gfCNCPoint3[24009] = {X 169.4126, Y 35.0505, Z -4.6667, A 0.000, B 0.000, C 0.000 }
gfCNCPoint3[24010] = {X 169.5555, Y 33.2588, Z -4.6667, A 0.000, B 0.000, C 0.000 }
gfCNCPoint3[24011] = {X 169.9217, Y 31.4991, Z -4.6667, A 0.000, B 0.000, C 0.000 }
gfCNCPoint3[24012] = {X 170.5055, Y 29.7991, Z -4.6667, A 0.000, B 0.000, C 0.000 }
gfCNCPoint3[24013] = {X 171.2083, Y 28.3890, Z -4.6667, A 0.000, B 0.000, C 0.000 }
gfCNCPoint3[24014] = {X 172.1134, Y 27.0994, Z -4.6667, A 0.000, B 0.000, C 0.000 }
gfCNCPoint3[24015] = {X 173.2007, Y 25.9592, Z -4.6667, A 0.000, B 0.000, C 0.000 }
gfCNCPoint3[24016] = {X 174.4459, Y 24.9938, Z -4.6667, A 0.000, B 0.000, C 0.000 }
gfCNCPoint3[24017] = {X 175.8210, Y 24.2248, Z -4.6667, A 0.000, B 0.000, C 0.000 }
gfCNCPoint3[24018] = {X 175.0301, Y 24.0138, Z -4.6667, A 0.000, B 0.000, C 0.000 }
gfCNCPoint3[24019] = {X 174.2987, Y 23.6462, Z -4.6667, A 0.000, B 0.000, C 0.000 }
gfCNCPoint3[24020] = {X 173.6575, Y 23.1374, Z -4.6667, A 0.000, B 0.000, C 0.000 }
gfCNCPoint3[24021] = {X 173.1332, Y 22.5088, Z -4.6667, A 0.000, B 0.000, C 0.000 }
gfCNCPoint3[24022] = {X 172.7479, Y 21.7866, Z -4.6667, A 0.000, B 0.000, C 0.000 }
gfCNCPoint3[24023] = {X 171.4542, Y 18.6179, Z -4.6667, A 0.000, B 0.000, C 0.000 }
gfCNCPoint3[24024] = {X 167.6769, Y 20.1601, Z -4.6667, A 0.000, B 0.000, C 0.000 }
gfCNCPoint3[24025] = {X 167.6769, Y 20.1601, Z -1.6667, A 0.000, B 0.000, C 0.000 }
gfCNCPoint3[24026] = {X 167.6769, Y 20.1601, Z 11.0000, A 0.000, B 0.000, C 0.000 }
gfCNCPoint3[24027] = {X 210.1649, Y 28.5740, Z 11.0000, A 0.000, B 0.000, C 0.000 }
gfCNCPoint3[24028] = {X 210.1649, Y 28.5740, Z -1.6667, A 0.000, B 0.000, C 0.000 }
gfCNCPoint3[24029] = {X 210.1649, Y 28.5740, Z -4.6667, A 0.000, B 0.000, C 0.000 }
gfCNCPoint3[24030] = {X 214.2449, Y 28.5740, Z -4.6667, A 0.000, B 0.000, C 0.000 }
gfCNCPoint3[24031] = {X 214.2449, Y 17.4625, Z -4.6667, A 0.000, B 0.000, C 0.000 }
gfCNCPoint3[24032] = {X 214.2395, Y 16.7693, Z -4.6667, A 0.000, B 0.000, C 0.000 }
gfCNCPoint3[24033] = {X 214.2427, Y 16.2726, Z -4.6667, A 0.000, B 0.000, C 0.000 }
gfCNCPoint3[24034] = {X 213.6048, Y 15.6014, Z -4.6667, A 0.000, B 0.000, C 0.000 }
gfCNCPoint3[24035] = {X 213.1246, Y 14.8098, Z -4.6667, A 0.000, B 0.000, C 0.000 }
gfCNCPoint3[24036] = {X 212.8241, Y 13.9340, Z -4.6667, A 0.000, B 0.000, C 0.000 }
gfCNCPoint3[24037] = {X 212.7172, Y 13.0143, Z -4.6667, A 0.000, B 0.000, C 0.000 }
gfCNCPoint3[24038] = {X 212.7170, Y 12.1868, Z -4.6667, A 0.000, B 0.000, C 0.000 }
gfCNCPoint3[24039] = {X 212.8253, Y 11.2255, Z -4.6667, A 0.000, B 0.000, C 0.000 }
gfCNCPoint3[24040] = {X 213.1448, Y 10.3124, Z -4.6667, A 0.000, B 0.000, C 0.000 }
gfCNCPoint3[24041] = {X 213.6595, Y 9.4933, Z -4.6667, A 0.000, B 0.000, C 0.000 }
gfCNCPoint3[24042] = {X 214.3435, Y 8.8093, Z -4.6667, A 0.000, B 0.000, C 0.000 }
gfCNCPoint3[24043] = {X 215.1626, Y 8.2946, Z -4.6667, A 0.000, B 0.000, C 0.000 }
gfCNCPoint3[24044] = {X 216.0757, Y 7.9751, Z -4.6667, A 0.000, B 0.000, C 0.000 }
gfCNCPoint3[24045] = {X 217.0370, Y 7.8668, Z -4.6667, A 0.000, B 0.000, C 0.000 }
gfCNCPoint3[24046] = {X 223.4805, Y 7.8668, Z -4.6667, A 0.000, B 0.000, C 0.000 }
gfCNCPoint3[24047] = {X 224.4418, Y 7.9751, Z -4.6667, A 0.000, B 0.000, C 0.000 }
gfCNCPoint3[24048] = {X 225.3549, Y 8.2946, Z -4.6667, A 0.000, B 0.000, C 0.000 }
gfCNCPoint3[24049] = {X 226.1740, Y 8.8093, Z -4.6667, A 0.000, B 0.000, C 0.000 }
gfCNCPoint3[24050] = {X 226.8580, Y 9.4933, Z -4.6667, A 0.000, B 0.000, C 0.000 }
gfCNCPoint3[24051] = {X 227.3727, Y 10.3124, Z -4.6667, A 0.000, B 0.000, C 0.000 }
gfCNCPoint3[24052] = {X 227.6922, Y 11.2255, Z -4.6667, A 0.000, B 0.000, C 0.000 }
gfCNCPoint3[24053] = {X 227.8005, Y 12.1868, Z -4.6667, A 0.000, B 0.000, C 0.000 }
gfCNCPoint3[24054] = {X 227.8005, Y 12.9782, Z -4.6667, A 0.000, B 0.000, C 0.000 }
gfCNCPoint3[24055] = {X 227.6992, Y 13.9081, Z -4.6667, A 0.000, B 0.000, C 0.000 }
gfCNCPoint3[24056] = {X 227.4001, Y 14.7944, Z -4.6667, A 0.000, B 0.000, C 0.000 }
gfCNCPoint3[24057] = {X 226.9172, Y 15.5955, Z -4.6667, A 0.000, B 0.000, C 0.000 }
gfCNCPoint3[24058] = {X 226.2732, Y 16.2739, Z -4.6667, A 0.000, B 0.000, C 0.000 }
gfCNCPoint3[24059] = {X 226.2742, Y 40.9155, Z -4.6667, A 0.000, B 0.000, C 0.000 }
gfCNCPoint3[24060] = {X 226.9115, Y 41.5856, Z -4.6667, A 0.000, B 0.000, C 0.000 }
gfCNCPoint3[24061] = {X 227.3916, Y 42.3760, Z -4.6667, A 0.000, B 0.000, C 0.000 }
gfCNCPoint3[24062] = {X 227.6924, Y 43.2504, Z -4.6667, A 0.000, B 0.000, C 0.000 }
gfCNCPoint3[24063] = {X 227.8003, Y 44.1689, Z -4.6667, A 0.000, B 0.000, C 0.000 }
gfCNCPoint3[24064] = {X 227.8005, Y 45.0000, Z -4.6667, A 0.000, B 0.000, C 0.000 }
gfCNCPoint3[24065] = {X 227.6922, Y 45.9613, Z -4.6667, A 0.000, B 0.000, C 0.000 }
gfCNCPoint3[24066] = {X 227.3727, Y 46.8744, Z -4.6667, A 0.000, B 0.000, C 0.000 }
gfCNCPoint3[24067] = {X 226.8580, Y 47.6935, Z -4.6667, A 0.000, B 0.000, C 0.000 }
gfCNCPoint3[24068] = {X 226.1740, Y 48.3775, Z -4.6667, A 0.000, B 0.000, C 0.000 }
gfCNCPoint3[24069] = {X 225.3549, Y 48.8922, Z -4.6667, A 0.000, B 0.000, C 0.000 }
gfCNCPoint3[24070] = {X 224.4418, Y 49.2117, Z -4.6667, A 0.000, B 0.000, C 0.000 }
gfCNCPoint3[24071] = {X 223.4805, Y 49.3200, Z -4.6667, A 0.000, B 0.000, C 0.000 }
gfCNCPoint3[24072] = {X 217.0370, Y 49.3200, Z -4.6667, A 0.000, B 0.000, C 0.000 }
gfCNCPoint3[24073] = {X 216.0805, Y 49.2128, Z -4.6667, A 0.000, B 0.000, C 0.000 }
gfCNCPoint3[24074] = {X 215.1715, Y 48.8964, Z -4.6667, A 0.000, B 0.000, C 0.000 }
gfCNCPoint3[24075] = {X 214.3551, Y 48.3867, Z -4.6667, A 0.000, B 0.000, C 0.000 }
gfCNCPoint3[24076] = {X 213.6718, Y 47.7088, Z -4.6667, A 0.000, B 0.000, C 0.000 }
gfCNCPoint3[24077] = {X 213.1556, Y 46.8965, Z -4.6667, A 0.000, B 0.000, C 0.000 }
gfCNCPoint3[24078] = {X 212.8320, Y 45.9901, Z -4.6667, A 0.000, B 0.000, C 0.000 }
gfCNCPoint3[24079] = {X 212.7172, Y 45.0345, Z -4.6667, A 0.000, B 0.000, C 0.000 }
gfCNCPoint3[24080] = {X 212.7170, Y 44.1958, Z -4.6667, A 0.000, B 0.000, C 0.000 }
gfCNCPoint3[24081] = {X 212.7889, Y 43.4176, Z -4.6667, A 0.000, B 0.000, C 0.000 }
gfCNCPoint3[24082] = {X 213.0019, Y 42.6657, Z -4.6667, A 0.000, B 0.000, C 0.000 }
gfCNCPoint3[24083] = {X 213.3491, Y 41.9656, Z -4.6667, A 0.000, B 0.000, C 0.000 }
gfCNCPoint3[24084] = {X 213.8185, Y 41.3408, Z -4.6667, A 0.000, B 0.000, C 0.000 }
gfCNCPoint3[24085] = {X 214.2405, Y 40.8754, Z -4.6667, A 0.000, B 0.000, C 0.000 }
gfCNCPoint3[24086] = {X 214.2449, Y 40.3061, Z -4.6667, A 0.000, B 0.000, C 0.000 }
gfCNCPoint3[24087] = {X 214.2449, Y 28.5740, Z -4.6667, A 0.000, B 0.000, C 0.000 }
gfCNCPoint3[24088] = {X 210.2449, Y 28.5740, Z -4.6667, A 0.000, B 0.000, C 0.000 }
gfCNCPoint3[24089] = {X 214.3249, Y 28.5740, Z -4.6667, A 0.000, B 0.000, C 0.000 }
gfCNCPoint3[24090] = {X 214.3249, Y 17.4621, Z -4.6667, A 0.000, B 0.000, C 0.000 }
gfCNCPoint3[24091] = {X 214.3195, Y 16.7692, Z -4.6667, A 0.000, B 0.000, C 0.000 }
gfCNCPoint3[24092] = {X 214.3229, Y 16.2355, Z -4.6667, A 0.000, B 0.000, C 0.000 }
gfCNCPoint3[24093] = {X 213.6854, Y 15.5750, Z -4.6667, A 0.000, B 0.000, C 0.000 }
gfCNCPoint3[24094] = {X 213.2050, Y 14.7927, Z -4.6667, A 0.000, B 0.000, C 0.000 }
gfCNCPoint3[24095] = {X 212.9042, Y 13.9254, Z -4.6667, A 0.000, B 0.000, C 0.000 }
gfCNCPoint3[24096] = {X 212.7972, Y 13.0137, Z -4.6667, A 0.000, B 0.000, C 0.000 }
gfCNCPoint3[24097] = {X 212.7970, Y 12.1868, Z -4.6667, A 0.000, B 0.000, C 0.000 }
gfCNCPoint3[24098] = {X 212.9033, Y 11.2433, Z -4.6667, A 0.000, B 0.000, C 0.000 }
gfCNCPoint3[24099] = {X 213.2169, Y 10.3472, Z -4.6667, A 0.000, B 0.000, C 0.000 }
gfCNCPoint3[24100] = {X 213.7220, Y 9.5432, Z -4.6667, A 0.000, B 0.000, C 0.000 }
gfCNCPoint3[24101] = {X 214.3934, Y 8.8719, Z -4.6667, A 0.000, B 0.000, C 0.000 }
gfCNCPoint3[24102] = {X 215.1973, Y 8.3667, Z -4.6667, A 0.000, B 0.000, C 0.000 }
gfCNCPoint3[24103] = {X 216.0935, Y 8.0531, Z -4.6667, A 0.000, B 0.000, C 0.000 }
gfCNCPoint3[24104] = {X 217.0370, Y 7.9468, Z -4.6667, A 0.000, B 0.000, C 0.000 }
gfCNCPoint3[24105] = {X 223.4805, Y 7.9468, Z -4.6667, A 0.000, B 0.000, C 0.000 }
gfCNCPoint3[24106] = {X 224.4240, Y 8.0531, Z -4.6667, A 0.000, B 0.000, C 0.000 }
gfCNCPoint3[24107] = {X 225.3201, Y 8.3667, Z -4.6667, A 0.000, B 0.000, C 0.000 }
gfCNCPoint3[24108] = {X 226.1241, Y 8.8718, Z -4.6667, A 0.000, B 0.000, C 0.000 }
gfCNCPoint3[24109] = {X 226.7954, Y 9.5432, Z -4.6667, A 0.000, B 0.000, C 0.000 }
gfCNCPoint3[24110] = {X 227.3006, Y 10.3471, Z -4.6667, A 0.000, B 0.000, C 0.000 }
gfCNCPoint3[24111] = {X 227.6142, Y 11.2433, Z -4.6667, A 0.000, B 0.000, C 0.000 }
gfCNCPoint3[24112] = {X 227.7205, Y 12.1868, Z -4.6667, A 0.000, B 0.000, C 0.000 }
gfCNCPoint3[24113] = {X 227.7205, Y 12.9781, Z -4.6667, A 0.000, B 0.000, C 0.000 }
gfCNCPoint3[24114] = {X 227.6191, Y 13.8998, Z -4.6667, A 0.000, B 0.000, C 0.000 }
gfCNCPoint3[24115] = {X 227.3197, Y 14.7775, Z -4.6667, A 0.000, B 0.000, C 0.000 }
gfCNCPoint3[24116] = {X 226.8367, Y 15.5690, Z -4.6667, A 0.000, B 0.000, C 0.000 }
gfCNCPoint3[24117] = {X 226.1932, Y 16.2366, Z -4.6667, A 0.000, B 0.000, C 0.000 }
gfCNCPoint3[24118] = {X 226.1942, Y 40.9527, Z -4.6667, A 0.000, B 0.000, C 0.000 }
gfCNCPoint3[24119] = {X 226.8310, Y 41.6122, Z -4.6667, A 0.000, B 0.000, C 0.000 }
gfCNCPoint3[24120] = {X 227.3113, Y 42.3932, Z -4.6667, A 0.000, B 0.000, C 0.000 }
gfCNCPoint3[24121] = {X 227.6124, Y 43.2592, Z -4.6667, A 0.000, B 0.000, C 0.000 }
gfCNCPoint3[24122] = {X 227.7203, Y 44.1697, Z -4.6667, A 0.000, B 0.000, C 0.000 }
gfCNCPoint3[24123] = {X 227.7205, Y 45.0000, Z -4.6667, A 0.000, B 0.000, C 0.000 }
gfCNCPoint3[24124] = {X 227.6142, Y 45.9435, Z -4.6667, A 0.000, B 0.000, C 0.000 }
gfCNCPoint3[24125] = {X 227.3006, Y 46.8397, Z -4.6667, A 0.000, B 0.000, C 0.000 }
gfCNCPoint3[24126] = {X 226.7954, Y 47.6436, Z -4.6667, A 0.000, B 0.000, C 0.000 }
gfCNCPoint3[24127] = {X 226.1241, Y 48.3150, Z -4.6667, A 0.000, B 0.000, C 0.000 }
gfCNCPoint3[24128] = {X 225.3201, Y 48.8201, Z -4.6667, A 0.000, B 0.000, C 0.000 }
gfCNCPoint3[24129] = {X 224.4240, Y 49.1337, Z -4.6667, A 0.000, B 0.000, C 0.000 }
gfCNCPoint3[24130] = {X 223.4805, Y 49.2400, Z -4.6667, A 0.000, B 0.000, C 0.000 }
gfCNCPoint3[24131] = {X 217.0370, Y 49.2400, Z -4.6667, A 0.000, B 0.000, C 0.000 }
gfCNCPoint3[24132] = {X 216.0982, Y 49.1348, Z -4.6667, A 0.000, B 0.000, C 0.000 }
gfCNCPoint3[24133] = {X 215.2061, Y 48.8243, Z -4.6667, A 0.000, B 0.000, C 0.000 }
gfCNCPoint3[24134] = {X 214.4048, Y 48.3240, Z -4.6667, A 0.000, B 0.000, C 0.000 }
gfCNCPoint3[24135] = {X 213.7341, Y 47.6587, Z -4.6667, A 0.000, B 0.000, C 0.000 }
gfCNCPoint3[24136] = {X 213.2275, Y 46.8614, Z -4.6667, A 0.000, B 0.000, C 0.000 }
gfCNCPoint3[24137] = {X 212.9099, Y 45.9717, Z -4.6667, A 0.000, B 0.000, C 0.000 }
gfCNCPoint3[24138] = {X 212.7972, Y 45.0338, Z -4.6667, A 0.000, B 0.000, C 0.000 }
gfCNCPoint3[24139] = {X 212.7970, Y 44.1958, Z -4.6667, A 0.000, B 0.000, C 0.000 }
gfCNCPoint3[24140] = {X 212.8675, Y 43.4322, Z -4.6667, A 0.000, B 0.000, C 0.000 }
gfCNCPoint3[24141] = {X 213.0766, Y 42.6945, Z -4.6667, A 0.000, B 0.000, C 0.000 }
gfCNCPoint3[24142] = {X 213.4172, Y 42.0076, Z -4.6667, A 0.000, B 0.000, C 0.000 }
gfCNCPoint3[24143] = {X 213.8778, Y 41.3946, Z -4.6667, A 0.000, B 0.000, C 0.000 }
gfCNCPoint3[24144] = {X 214.3203, Y 40.9065, Z -4.6667, A 0.000, B 0.000, C 0.000 }
gfCNCPoint3[24145] = {X 214.3249, Y 40.3065, Z -4.6667, A 0.000, B 0.000, C 0.000 }
gfCNCPoint3[24146] = {X 214.3249, Y 28.5740, Z -4.6667, A 0.000, B 0.000, C 0.000 }
gfCNCPoint3[24147] = {X 210.3249, Y 28.5740, Z -4.6667, A 0.000, B 0.000, C 0.000 }
gfCNCPoint3[24148] = {X 214.4049, Y 28.5740, Z -4.6667, A 0.000, B 0.000, C 0.000 }
gfCNCPoint3[24149] = {X 214.4049, Y 17.4618, Z -4.6667, A 0.000, B 0.000, C 0.000 }
gfCNCPoint3[24150] = {X 214.3995, Y 16.7691, Z -4.6667, A 0.000, B 0.000, C 0.000 }
gfCNCPoint3[24151] = {X 214.4031, Y 16.1980, Z -4.6667, A 0.000, B 0.000, C 0.000 }
gfCNCPoint3[24152] = {X 213.7660, Y 15.5482, Z -4.6667, A 0.000, B 0.000, C 0.000 }
gfCNCPoint3[24153] = {X 213.2854, Y 14.7755, Z -4.6667, A 0.000, B 0.000, C 0.000 }
gfCNCPoint3[24154] = {X 212.9843, Y 13.9167, Z -4.6667, A 0.000, B 0.000, C 0.000 }
gfCNCPoint3[24155] = {X 212.8772, Y 13.0130, Z -4.6667, A 0.000, B 0.000, C 0.000 }
gfCNCPoint3[24156] = {X 212.8770, Y 12.1868, Z -4.6667, A 0.000, B 0.000, C 0.000 }
gfCNCPoint3[24157] = {X 212.9813, Y 11.2611, Z -4.6667, A 0.000, B 0.000, C 0.000 }
gfCNCPoint3[24158] = {X 213.2890, Y 10.3819, Z -4.6667, A 0.000, B 0.000, C 0.000 }
gfCNCPoint3[24159] = {X 213.7846, Y 9.5931, Z -4.6667, A 0.000, B 0.000, C 0.000 }
gfCNCPoint3[24160] = {X 214.4433, Y 8.9344, Z -4.6667, A 0.000, B 0.000, C 0.000 }
gfCNCPoint3[24161] = {X 215.2321, Y 8.4388, Z -4.6667, A 0.000, B 0.000, C 0.000 }
gfCNCPoint3[24162] = {X 216.1113, Y 8.1311, Z -4.6667, A 0.000, B 0.000, C 0.000 }
gfCNCPoint3[24163] = {X 217.0370, Y 8.0268, Z -4.6667, A 0.000, B 0.000, C 0.000 }
gfCNCPoint3[24164] = {X 223.4805, Y 8.0268, Z -4.6667, A 0.000, B 0.000, C 0.000 }
gfCNCPoint3[24165] = {X 224.4062, Y 8.1311, Z -4.6667, A 0.000, B 0.000, C 0.000 }
gfCNCPoint3[24166] = {X 225.2854, Y 8.4388, Z -4.6667, A 0.000, B 0.000, C 0.000 }
gfCNCPoint3[24167] = {X 226.0742, Y 8.9344, Z -4.6667, A 0.000, B 0.000, C 0.000 }
gfCNCPoint3[24168] = {X 226.7329, Y 9.5931, Z -4.6667, A 0.000, B 0.000, C 0.000 }
gfCNCPoint3[24169] = {X 227.2285, Y 10.3819, Z -4.6667, A 0.000, B 0.000, C 0.000 }
gfCNCPoint3[24170] = {X 227.5362, Y 11.2611, Z -4.6667, A 0.000, B 0.000, C 0.000 }
gfCNCPoint3[24171] = {X 227.6405, Y 12.1868, Z -4.6667, A 0.000, B 0.000, C 0.000 }
gfCNCPoint3[24172] = {X 227.6405, Y 12.9781, Z -4.6667, A 0.000, B 0.000, C 0.000 }
gfCNCPoint3[24173] = {X 227.5389, Y 13.8916, Z -4.6667, A 0.000, B 0.000, C 0.000 }
gfCNCPoint3[24174] = {X 227.2393, Y 14.7604, Z -4.6667, A 0.000, B 0.000, C 0.000 }
gfCNCPoint3[24175] = {X 226.7562, Y 15.5422, Z -4.6667, A 0.000, B 0.000, C 0.000 }
gfCNCPoint3[24176] = {X 226.1132, Y 16.1989, Z -4.6667, A 0.000, B 0.000, C 0.000 }
gfCNCPoint3[24177] = {X 226.1142, Y 40.9904, Z -4.6667, A 0.000, B 0.000, C 0.000 }
gfCNCPoint3[24178] = {X 226.7506, Y 41.6392, Z -4.6667, A 0.000, B 0.000, C 0.000 }
gfCNCPoint3[24179] = {X 227.2310, Y 42.4107, Z -4.6667, A 0.000, B 0.000, C 0.000 }
gfCNCPoint3[24180] = {X 227.5323, Y 43.2681, Z -4.6667, A 0.000, B 0.000, C 0.000 }
gfCNCPoint3[24181] = {X 227.6403, Y 44.1704, Z -4.6667, A 0.000, B 0.000, C 0.000 }
gfCNCPoint3[24182] = {X 227.6405, Y 45.0000, Z -4.6667, A 0.000, B 0.000, C 0.000 }
gfCNCPoint3[24183] = {X 227.5362, Y 45.9257, Z -4.6667, A 0.000, B 0.000, C 0.000 }
gfCNCPoint3[24184] = {X 227.2285, Y 46.8050, Z -4.6667, A 0.000, B 0.000, C 0.000 }
gfCNCPoint3[24185] = {X 226.7329, Y 47.5937, Z -4.6667, A 0.000, B 0.000, C 0.000 }
gfCNCPoint3[24186] = {X 226.0742, Y 48.2524, Z -4.6667, A 0.000, B 0.000, C 0.000 }
gfCNCPoint3[24187] = {X 225.2854, Y 48.7480, Z -4.6667, A 0.000, B 0.000, C 0.000 }
gfCNCPoint3[24188] = {X 224.4062, Y 49.0557, Z -4.6667, A 0.000, B 0.000, C 0.000 }
gfCNCPoint3[24189] = {X 223.4805, Y 49.1600, Z -4.6667, A 0.000, B 0.000, C 0.000 }
gfCNCPoint3[24190] = {X 217.0370, Y 49.1600, Z -4.6667, A 0.000, B 0.000, C 0.000 }
gfCNCPoint3[24191] = {X 216.1160, Y 49.0568, Z -4.6667, A 0.000, B 0.000, C 0.000 }
gfCNCPoint3[24192] = {X 215.2406, Y 48.7521, Z -4.6667, A 0.000, B 0.000, C 0.000 }
gfCNCPoint3[24193] = {X 214.4544, Y 48.2613, Z -4.6667, A 0.000, B 0.000, C 0.000 }
gfCNCPoint3[24194] = {X 213.7965, Y 47.6085, Z -4.6667, A 0.000, B 0.000, C 0.000 }
gfCNCPoint3[24195] = {X 213.2993, Y 46.8263, Z -4.6667, A 0.000, B 0.000, C 0.000 }
gfCNCPoint3[24196] = {X 212.9877, Y 45.9534, Z -4.6667, A 0.000, B 0.000, C 0.000 }
gfCNCPoint3[24197] = {X 212.8771, Y 45.0332, Z -4.6667, A 0.000, B 0.000, C 0.000 }
gfCNCPoint3[24198] = {X 212.8770, Y 44.1958, Z -4.6667, A 0.000, B 0.000, C 0.000 }
gfCNCPoint3[24199] = {X 212.9461, Y 43.4469, Z -4.6667, A 0.000, B 0.000, C 0.000 }
gfCNCPoint3[24200] = {X 213.1512, Y 42.7233, Z -4.6667, A 0.000, B 0.000, C 0.000 }
gfCNCPoint3[24201] = {X 213.4853, Y 42.0495, Z -4.6667, A 0.000, B 0.000, C 0.000 }
gfCNCPoint3[24202] = {X 213.9370, Y 41.4483, Z -4.6667, A 0.000, B 0.000, C 0.000 }
gfCNCPoint3[24203] = {X 214.4000, Y 40.9376, Z -4.6667, A 0.000, B 0.000, C 0.000 }
gfCNCPoint3[24204] = {X 214.4049, Y 40.3068, Z -4.6667, A 0.000, B 0.000, C 0.000 }
gfCNCPoint3[24205] = {X 214.4049, Y 28.5740, Z -4.6667, A 0.000, B 0.000, C 0.000 }
gfCNCPoint3[24206] = {X 210.4049, Y 28.5740, Z -4.6667, A 0.000, B 0.000, C 0.000 }
gfCNCPoint3[24207] = {X 214.4849, Y 28.5740, Z -4.6667, A 0.000, B 0.000, C 0.000 }
gfCNCPoint3[24208] = {X 214.4849, Y 17.4614, Z -4.6667, A 0.000, B 0.000, C 0.000 }
gfCNCPoint3[24209] = {X 214.4795, Y 16.7691, Z -4.6667, A 0.000, B 0.000, C 0.000 }
gfCNCPoint3[24210] = {X 214.4834, Y 16.1601, Z -4.6667, A 0.000, B 0.000, C 0.000 }
gfCNCPoint3[24211] = {X 214.4254, Y 16.1127, Z -4.6667, A 0.000, B 0.000, C 0.000 }
gfCNCPoint3[24212] = {X 214.3684, Y 16.0642, Z -4.6667, A 0.000, B 0.000, C 0.000 }
gfCNCPoint3[24213] = {X 213.7778, Y 15.4325, Z -4.6667, A 0.000, B 0.000, C 0.000 }
gfCNCPoint3[24214] = {X 213.3338, Y 14.6904, Z -4.6667, A 0.000, B 0.000, C 0.000 }
gfCNCPoint3[24215] = {X 213.0560, Y 13.8714, Z -4.6667, A 0.000, B 0.000, C 0.000 }
gfCNCPoint3[24216] = {X 212.9572, Y 13.0123, Z -4.6667, A 0.000, B 0.000, C 0.000 }
gfCNCPoint3[24217] = {X 212.9570, Y 12.1868, Z -4.6667, A 0.000, B 0.000, C 0.000 }
gfCNCPoint3[24218] = {X 213.0593, Y 11.2789, Z -4.6667, A 0.000, B 0.000, C 0.000 }
gfCNCPoint3[24219] = {X 213.3611, Y 10.4166, Z -4.6667, A 0.000, B 0.000, C 0.000 }
gfCNCPoint3[24220] = {X 213.8471, Y 9.6430, Z -4.6667, A 0.000, B 0.000, C 0.000 }
gfCNCPoint3[24221] = {X 214.4932, Y 8.9969, Z -4.6667, A 0.000, B 0.000, C 0.000 }
gfCNCPoint3[24222] = {X 215.2668, Y 8.5109, Z -4.6667, A 0.000, B 0.000, C 0.000 }
gfCNCPoint3[24223] = {X 216.1291, Y 8.2091, Z -4.6667, A 0.000, B 0.000, C 0.000 }
gfCNCPoint3[24224] = {X 217.0370, Y 8.1068, Z -4.6667, A 0.000, B 0.000, C 0.000 }
gfCNCPoint3[24225] = {X 223.4805, Y 8.1068, Z -4.6667, A 0.000, B 0.000, C 0.000 }
gfCNCPoint3[24226] = {X 224.3884, Y 8.2091, Z -4.6667, A 0.000, B 0.000, C 0.000 }
gfCNCPoint3[24227] = {X 225.2507, Y 8.5109, Z -4.6667, A 0.000, B 0.000, C 0.000 }
gfCNCPoint3[24228] = {X 226.0243, Y 8.9969, Z -4.6667, A 0.000, B 0.000, C 0.000 }
gfCNCPoint3[24229] = {X 226.6704, Y 9.6430, Z -4.6667, A 0.000, B 0.000, C 0.000 }
gfCNCPoint3[24230] = {X 227.1564, Y 10.4166, Z -4.6667, A 0.000, B 0.000, C 0.000 }
gfCNCPoint3[24231] = {X 227.4582, Y 11.2789, Z -4.6667, A 0.000, B 0.000, C 0.000 }
gfCNCPoint3[24232] = {X 227.5605, Y 12.1868, Z -4.6667, A 0.000, B 0.000, C 0.000 }
gfCNCPoint3[24233] = {X 227.5605, Y 12.9781, Z -4.6667, A 0.000, B 0.000, C 0.000 }
gfCNCPoint3[24234] = {X 227.4588, Y 13.8832, Z -4.6667, A 0.000, B 0.000, C 0.000 }
gfCNCPoint3[24235] = {X 227.1589, Y 14.7432, Z -4.6667, A 0.000, B 0.000, C 0.000 }
gfCNCPoint3[24236] = {X 226.6757, Y 15.5152, Z -4.6667, A 0.000, B 0.000, C 0.000 }
gfCNCPoint3[24237] = {X 226.0332, Y 16.1608, Z -4.6667, A 0.000, B 0.000, C 0.000 }
gfCNCPoint3[24238] = {X 226.0342, Y 41.0284, Z -4.6667, A 0.000, B 0.000, C 0.000 }
gfCNCPoint3[24239] = {X 226.1410, Y 41.1156, Z -4.6667, A 0.000, B 0.000, C 0.000 }
gfCNCPoint3[24240] = {X 226.7343, Y 41.7473, Z -4.6667, A 0.000, B 0.000, C 0.000 }
gfCNCPoint3[24241] = {X 227.1808, Y 42.4900, Z -4.6667, A 0.000, B 0.000, C 0.000 }
gfCNCPoint3[24242] = {X 227.4603, Y 43.3103, Z -4.6667, A 0.000, B 0.000, C 0.000 }
gfCNCPoint3[24243] = {X 227.5603, Y 44.1712, Z -4.6667, A 0.000, B 0.000, C 0.000 }
gfCNCPoint3[24244] = {X 227.5605, Y 45.0000, Z -4.6667, A 0.000, B 0.000, C 0.000 }
gfCNCPoint3[24245] = {X 227.4582, Y 45.9079, Z -4.6667, A 0.000, B 0.000, C 0.000 }
gfCNCPoint3[24246] = {X 227.1564, Y 46.7702, Z -4.6667, A 0.000, B 0.000, C 0.000 }
gfCNCPoint3[24247] = {X 226.6704, Y 47.5438, Z -4.6667, A 0.000, B 0.000, C 0.000 }
gfCNCPoint3[24248] = {X 226.0243, Y 48.1899, Z -4.6667, A 0.000, B 0.000, C 0.000 }
gfCNCPoint3[24249] = {X 225.2507, Y 48.6760, Z -4.6667, A 0.000, B 0.000, C 0.000 }
gfCNCPoint3[24250] = {X 224.3884, Y 48.9777, Z -4.6667, A 0.000, B 0.000, C 0.000 }
gfCNCPoint3[24251] = {X 223.4805, Y 49.0800, Z -4.6667, A 0.000, B 0.000, C 0.000 }
gfCNCPoint3[24252] = {X 217.0370, Y 49.0800, Z -4.6667, A 0.000, B 0.000, C 0.000 }
gfCNCPoint3[24253] = {X 216.1337, Y 48.9787, Z -4.6667, A 0.000, B 0.000, C 0.000 }
gfCNCPoint3[24254] = {X 215.2752, Y 48.6800, Z -4.6667, A 0.000, B 0.000, C 0.000 }
gfCNCPoint3[24255] = {X 214.5041, Y 48.1986, Z -4.6667, A 0.000, B 0.000, C 0.000 }
gfCNCPoint3[24256] = {X 213.8588, Y 47.5584, Z -4.6667, A 0.000, B 0.000, C 0.000 }
gfCNCPoint3[24257] = {X 213.3712, Y 46.7912, Z -4.6667, A 0.000, B 0.000, C 0.000 }
gfCNCPoint3[24258] = {X 213.0656, Y 45.9351, Z -4.6667, A 0.000, B 0.000, C 0.000 }
gfCNCPoint3[24259] = {X 212.9571, Y 45.0325, Z -4.6667, A 0.000, B 0.000, C 0.000 }
gfCNCPoint3[24260] = {X 212.9570, Y 44.1958, Z -4.6667, A 0.000, B 0.000, C 0.000 }
gfCNCPoint3[24261] = {X 213.0248, Y 43.4615, Z -4.6667, A 0.000, B 0.000, C 0.000 }
gfCNCPoint3[24262] = {X 213.2259, Y 42.7521, Z -4.6667, A 0.000, B 0.000, C 0.000 }
gfCNCPoint3[24263] = {X 213.5534, Y 42.0915, Z -4.6667, A 0.000, B 0.000, C 0.000 }
gfCNCPoint3[24264] = {X 213.9963, Y 41.5020, Z -4.6667, A 0.000, B 0.000, C 0.000 }
gfCNCPoint3[24265] = {X 214.4798, Y 40.9687, Z -4.6667, A 0.000, B 0.000, C 0.000 }
gfCNCPoint3[24266] = {X 214.4849, Y 40.3072, Z -4.6667, A 0.000, B 0.000, C 0.000 }
gfCNCPoint3[24267] = {X 214.4849, Y 28.5740, Z -4.6667, A 0.000, B 0.000, C 0.000 }
gfCNCPoint3[24268] = {X 210.4849, Y 28.5740, Z -4.6667, A 0.000, B 0.000, C 0.000 }
gfCNCPoint3[24269] = {X 214.5649, Y 28.5740, Z -4.6667, A 0.000, B 0.000, C 0.000 }
gfCNCPoint3[24270] = {X 214.5649, Y 17.4611, Z -4.6667, A 0.000, B 0.000, C 0.000 }
gfCNCPoint3[24271] = {X 214.5595, Y 16.7687, Z -4.6667, A 0.000, B 0.000, C 0.000 }
gfCNCPoint3[24272] = {X 214.5589, Y 16.1867, Z -4.6667, A 0.000, B 0.000, C 0.000 }
gfCNCPoint3[24273] = {X 214.5756, Y 16.1310, Z -4.6667, A 0.000, B 0.000, C 0.000 }
gfCNCPoint3[24274] = {X 214.4973, Y 16.0683, Z -4.6667, A 0.000, B 0.000, C 0.000 }
gfCNCPoint3[24275] = {X 214.4207, Y 16.0037, Z -4.6667, A 0.000, B 0.000, C 0.000 }
gfCNCPoint3[24276] = {X 213.8367, Y 15.3776, Z -4.6667, A 0.000, B 0.000, C 0.000 }
gfCNCPoint3[24277] = {X 213.3993, Y 14.6415, Z -4.6667, A 0.000, B 0.000, C 0.000 }
gfCNCPoint3[24278] = {X 213.1286, Y 13.8292, Z -4.6667, A 0.000, B 0.000, C 0.000 }
gfCNCPoint3[24279] = {X 213.0370, Y 12.9779, Z -4.6667, A 0.000, B 0.000, C 0.000 }
gfCNCPoint3[24280] = {X 213.0370, Y 12.1868, Z -4.6667, A 0.000, B 0.000, C 0.000 }
gfCNCPoint3[24281] = {X 213.1373, Y 11.2967, Z -4.6667, A 0.000, B 0.000, C 0.000 }
gfCNCPoint3[24282] = {X 213.4331, Y 10.4513, Z -4.6667, A 0.000, B 0.000, C 0.000 }
gfCNCPoint3[24283] = {X 213.9097, Y 9.6929, Z -4.6667, A 0.000, B 0.000, C 0.000 }
gfCNCPoint3[24284] = {X 214.5431, Y 9.0595, Z -4.6667, A 0.000, B 0.000, C 0.000 }
gfCNCPoint3[24285] = {X 215.3015, Y 8.5829, Z -4.6667, A 0.000, B 0.000, C 0.000 }
gfCNCPoint3[24286] = {X 216.1469, Y 8.2871, Z -4.6667, A 0.000, B 0.000, C 0.000 }
gfCNCPoint3[24287] = {X 217.0370, Y 8.1868, Z -4.6667, A 0.000, B 0.000, C 0.000 }
gfCNCPoint3[24288] = {X 223.4805, Y 8.1868, Z -4.6667, A 0.000, B 0.000, C 0.000 }
gfCNCPoint3[24289] = {X 224.3706, Y 8.2871, Z -4.6667, A 0.000, B 0.000, C 0.000 }
gfCNCPoint3[24290] = {X 225.2160, Y 8.5829, Z -4.6667, A 0.000, B 0.000, C 0.000 }
gfCNCPoint3[24291] = {X 225.9744, Y 9.0595, Z -4.6667, A 0.000, B 0.000, C 0.000 }
gfCNCPoint3[24292] = {X 226.6078, Y 9.6929, Z -4.6667, A 0.000, B 0.000, C 0.000 }
gfCNCPoint3[24293] = {X 227.0844, Y 10.4513, Z -4.6667, A 0.000, B 0.000, C 0.000 }
gfCNCPoint3[24294] = {X 227.3802, Y 11.2967, Z -4.6667, A 0.000, B 0.000, C 0.000 }
gfCNCPoint3[24295] = {X 227.4805, Y 12.1868, Z -4.6667, A 0.000, B 0.000, C 0.000 }
gfCNCPoint3[24296] = {X 227.4803, Y 13.0192, Z -4.6667, A 0.000, B 0.000, C 0.000 }
gfCNCPoint3[24297] = {X 227.3716, Y 13.9048, Z -4.6667, A 0.000, B 0.000, C 0.000 }
gfCNCPoint3[24298] = {X 227.0694, Y 14.7442, Z -4.6667, A 0.000, B 0.000, C 0.000 }
gfCNCPoint3[24299] = {X 226.5887, Y 15.4958, Z -4.6667, A 0.000, B 0.000, C 0.000 }
gfCNCPoint3[24300] = {X 225.9532, Y 16.1221, Z -4.6667, A 0.000, B 0.000, C 0.000 }
gfCNCPoint3[24301] = {X 225.9542, Y 41.0664, Z -4.6667, A 0.000, B 0.000, C 0.000 }
gfCNCPoint3[24302] = {X 226.0929, Y 41.1797, Z -4.6667, A 0.000, B 0.000, C 0.000 }
gfCNCPoint3[24303] = {X 226.6785, Y 41.8061, Z -4.6667, A 0.000, B 0.000, C 0.000 }
gfCNCPoint3[24304] = {X 227.1171, Y 42.5430, Z -4.6667, A 0.000, B 0.000, C 0.000 }
gfCNCPoint3[24305] = {X 227.3886, Y 43.3563, Z -4.6667, A 0.000, B 0.000, C 0.000 }
gfCNCPoint3[24306] = {X 227.4805, Y 44.2089, Z -4.6667, A 0.000, B 0.000, C 0.000 }
gfCNCPoint3[24307] = {X 227.4805, Y 45.0000, Z -4.6667, A 0.000, B 0.000, C 0.000 }
gfCNCPoint3[24308] = {X 227.3802, Y 45.8901, Z -4.6667, A 0.000, B 0.000, C 0.000 }
gfCNCPoint3[24309] = {X 227.0844, Y 46.7355, Z -4.6667, A 0.000, B 0.000, C 0.000 }
gfCNCPoint3[24310] = {X 226.6078, Y 47.4940, Z -4.6667, A 0.000, B 0.000, C 0.000 }
gfCNCPoint3[24311] = {X 225.9744, Y 48.1273, Z -4.6667, A 0.000, B 0.000, C 0.000 }
gfCNCPoint3[24312] = {X 225.2160, Y 48.6039, Z -4.6667, A 0.000, B 0.000, C 0.000 }
gfCNCPoint3[24313] = {X 224.3706, Y 48.8997, Z -4.6667, A 0.000, B 0.000, C 0.000 }
gfCNCPoint3[24314] = {X 223.4805, Y 49.0000, Z -4.6667, A 0.000, B 0.000, C 0.000 }
gfCNCPoint3[24315] = {X 217.0370, Y 49.0000, Z -4.6667, A 0.000, B 0.000, C 0.000 }
gfCNCPoint3[24316] = {X 216.1469, Y 48.8997, Z -4.6667, A 0.000, B 0.000, C 0.000 }
gfCNCPoint3[24317] = {X 215.3015, Y 48.6039, Z -4.6667, A 0.000, B 0.000, C 0.000 }
gfCNCPoint3[24318] = {X 214.5430, Y 48.1273, Z -4.6667, A 0.000, B 0.000, C 0.000 }
gfCNCPoint3[24319] = {X 213.9097, Y 47.4939, Z -4.6667, A 0.000, B 0.000, C 0.000 }
gfCNCPoint3[24320] = {X 213.4331, Y 46.7355, Z -4.6667, A 0.000, B 0.000, C 0.000 }
gfCNCPoint3[24321] = {X 213.1373, Y 45.8901, Z -4.6667, A 0.000, B 0.000, C 0.000 }
gfCNCPoint3[24322] = {X 213.0370, Y 45.0000, Z -4.6667, A 0.000, B 0.000, C 0.000 }
gfCNCPoint3[24323] = {X 213.0370, Y 44.1958, Z -4.6667, A 0.000, B 0.000, C 0.000 }
gfCNCPoint3[24324] = {X 213.1549, Y 43.2405, Z -4.6667, A 0.000, B 0.000, C 0.000 }
gfCNCPoint3[24325] = {X 213.5013, Y 42.3426, Z -4.6667, A 0.000, B 0.000, C 0.000 }
gfCNCPoint3[24326] = {X 214.0556, Y 41.5557, Z -4.6667, A 0.000, B 0.000, C 0.000 }
gfCNCPoint3[24327] = {X 214.5595, Y 40.9999, Z -4.6667, A 0.000, B 0.000, C 0.000 }
gfCNCPoint3[24328] = {X 214.5649, Y 40.3075, Z -4.6667, A 0.000, B 0.000, C 0.000 }
gfCNCPoint3[24329] = {X 214.5649, Y 28.5740, Z -4.6667, A 0.000, B 0.000, C 0.000 }
gfCNCPoint3[24330] = {X 210.4849, Y 28.5740, Z -4.6667, A 0.000, B 0.000, C 0.000 }
gfCNCPoint3[24331] = {X 210.4849, Y 28.5740, Z -1.6667, A 0.000, B 0.000, C 0.000 }
gfCNCPoint3[24332] = {X 210.4849, Y 28.5740, Z 11.0000, A 0.000, B 0.000, C 0.000 }
gfCNCPoint3[24333] = {X 273.6039, Y 28.5936, Z 11.0000, A 0.000, B 0.000, C 0.000 }
gfCNCPoint3[24334] = {X 273.6039, Y 28.5936, Z -1.6667, A 0.000, B 0.000, C 0.000 }
gfCNCPoint3[24335] = {X 273.6039, Y 28.5936, Z -4.6667, A 0.000, B 0.000, C 0.000 }
gfCNCPoint3[24336] = {X 269.5239, Y 28.5936, Z -4.6667, A 0.000, B 0.000, C 0.000 }
gfCNCPoint3[24337] = {X 269.5239, Y 40.9135, Z -4.6667, A 0.000, B 0.000, C 0.000 }
gfCNCPoint3[24338] = {X 269.5375, Y 40.9245, Z -4.6667, A 0.000, B 0.000, C 0.000 }
gfCNCPoint3[24339] = {X 270.1699, Y 41.5940, Z -4.6667, A 0.000, B 0.000, C 0.000 }
gfCNCPoint3[24340] = {X 270.6460, Y 42.3824, Z -4.6667, A 0.000, B 0.000, C 0.000 }
gfCNCPoint3[24341] = {X 270.9441, Y 43.2538, Z -4.6667, A 0.000, B 0.000, C 0.000 }
gfCNCPoint3[24342] = {X 271.0508, Y 44.1686, Z -4.6667, A 0.000, B 0.000, C 0.000 }
gfCNCPoint3[24343] = {X 271.0510, Y 45.0000, Z -4.6667, A 0.000, B 0.000, C 0.000 }
gfCNCPoint3[24344] = {X 270.9427, Y 45.9613, Z -4.6667, A 0.000, B 0.000, C 0.000 }
gfCNCPoint3[24345] = {X 270.6232, Y 46.8744, Z -4.6667, A 0.000, B 0.000, C 0.000 }
gfCNCPoint3[24346] = {X 270.1085, Y 47.6935, Z -4.6667, A 0.000, B 0.000, C 0.000 }
gfCNCPoint3[24347] = {X 269.4245, Y 48.3775, Z -4.6667, A 0.000, B 0.000, C 0.000 }
gfCNCPoint3[24348] = {X 268.6054, Y 48.8922, Z -4.6667, A 0.000, B 0.000, C 0.000 }
gfCNCPoint3[24349] = {X 267.6923, Y 49.2117, Z -4.6667, A 0.000, B 0.000, C 0.000 }
gfCNCPoint3[24350] = {X 266.7310, Y 49.3200, Z -4.6667, A 0.000, B 0.000, C 0.000 }
gfCNCPoint3[24351] = {X 260.2876, Y 49.3200, Z -4.6667, A 0.000, B 0.000, C 0.000 }
gfCNCPoint3[24352] = {X 259.3310, Y 49.2128, Z -4.6667, A 0.000, B 0.000, C 0.000 }
gfCNCPoint3[24353] = {X 258.4219, Y 48.8963, Z -4.6667, A 0.000, B 0.000, C 0.000 }
gfCNCPoint3[24354] = {X 257.6054, Y 48.3865, Z -4.6667, A 0.000, B 0.000, C 0.000 }
gfCNCPoint3[24355] = {X 256.9221, Y 47.7085, Z -4.6667, A 0.000, B 0.000, C 0.000 }
gfCNCPoint3[24356] = {X 256.4059, Y 46.8960, Z -4.6667, A 0.000, B 0.000, C 0.000 }
gfCNCPoint3[24357] = {X 256.0824, Y 45.9894, Z -4.6667, A 0.000, B 0.000, C 0.000 }
gfCNCPoint3[24358] = {X 255.9677, Y 45.0336, Z -4.6667, A 0.000, B 0.000, C 0.000 }
gfCNCPoint3[24359] = {X 255.9680, Y 44.1494, Z -4.6667, A 0.000, B 0.000, C 0.000 }
gfCNCPoint3[24360] = {X 256.0784, Y 43.2364, Z -4.6667, A 0.000, B 0.000, C 0.000 }
gfCNCPoint3[24361] = {X 256.3796, Y 42.3675, Z -4.6667, A 0.000, B 0.000, C 0.000 }
gfCNCPoint3[24362] = {X 256.8579, Y 41.5821, Z -4.6667, A 0.000, B 0.000, C 0.000 }
gfCNCPoint3[24363] = {X 257.4915, Y 40.9157, Z -4.6667, A 0.000, B 0.000, C 0.000 }
gfCNCPoint3[24364] = {X 257.4915, Y 34.4738, Z -4.6667, A 0.000, B 0.000, C 0.000 }
gfCNCPoint3[24365] = {X 254.7677, Y 34.4738, Z -4.6667, A 0.000, B 0.000, C 0.000 }
gfCNCPoint3[24366] = {X 250.4838, Y 42.8186, Z -4.6667, A 0.000, B 0.000, C 0.000 }
gfCNCPoint3[24367] = {X 250.6527, Y 43.4863, Z -4.6667, A 0.000, B 0.000, C 0.000 }
gfCNCPoint3[24368] = {X 250.7134, Y 44.1723, Z -4.6667, A 0.000, B 0.000, C 0.000 }
gfCNCPoint3[24369] = {X 250.7136, Y 45.0000, Z -4.6667, A 0.000, B 0.000, C 0.000 }
gfCNCPoint3[24370] = {X 250.6052, Y 45.9613, Z -4.6667, A 0.000, B 0.000, C 0.000 }
gfCNCPoint3[24371] = {X 250.2857, Y 46.8744, Z -4.6667, A 0.000, B 0.000, C 0.000 }
gfCNCPoint3[24372] = {X 249.7711, Y 47.6935, Z -4.6667, A 0.000, B 0.000, C 0.000 }
gfCNCPoint3[24373] = {X 249.0870, Y 48.3775, Z -4.6667, A 0.000, B 0.000, C 0.000 }
gfCNCPoint3[24374] = {X 248.2679, Y 48.8922, Z -4.6667, A 0.000, B 0.000, C 0.000 }
gfCNCPoint3[24375] = {X 247.3548, Y 49.2117, Z -4.6667, A 0.000, B 0.000, C 0.000 }
gfCNCPoint3[24376] = {X 246.3936, Y 49.3200, Z -4.6667, A 0.000, B 0.000, C 0.000 }
gfCNCPoint3[24377] = {X 239.8075, Y 49.3200, Z -4.6667, A 0.000, B 0.000, C 0.000 }
gfCNCPoint3[24378] = {X 238.8462, Y 49.2117, Z -4.6667, A 0.000, B 0.000, C 0.000 }
gfCNCPoint3[24379] = {X 237.9331, Y 48.8922, Z -4.6667, A 0.000, B 0.000, C 0.000 }
gfCNCPoint3[24380] = {X 237.1141, Y 48.3775, Z -4.6667, A 0.000, B 0.000, C 0.000 }
gfCNCPoint3[24381] = {X 236.4300, Y 47.6935, Z -4.6667, A 0.000, B 0.000, C 0.000 }
gfCNCPoint3[24382] = {X 235.9153, Y 46.8745, Z -4.6667, A 0.000, B 0.000, C 0.000 }
gfCNCPoint3[24383] = {X 235.5958, Y 45.9614, Z -4.6667, A 0.000, B 0.000, C 0.000 }
gfCNCPoint3[24384] = {X 235.4875, Y 45.0001, Z -4.6667, A 0.000, B 0.000, C 0.000 }
gfCNCPoint3[24385] = {X 235.4879, Y 44.1494, Z -4.6667, A 0.000, B 0.000, C 0.000 }
gfCNCPoint3[24386] = {X 235.5856, Y 43.2935, Z -4.6667, A 0.000, B 0.000, C 0.000 }
gfCNCPoint3[24387] = {X 235.8511, Y 42.4740, Z -4.6667, A 0.000, B 0.000, C 0.000 }
gfCNCPoint3[24388] = {X 236.2739, Y 41.7236, Z -4.6667, A 0.000, B 0.000, C 0.000 }
gfCNCPoint3[24389] = {X 236.8373, Y 41.0719, Z -4.6667, A 0.000, B 0.000, C 0.000 }
gfCNCPoint3[24390] = {X 237.5187, Y 40.5449, Z -4.6667, A 0.000, B 0.000, C 0.000 }
gfCNCPoint3[24391] = {X 238.2911, Y 40.1637, Z -4.6667, A 0.000, B 0.000, C 0.000 }
gfCNCPoint3[24392] = {X 242.2803, Y 32.3554, Z -4.6667, A 0.000, B 0.000, C 0.000 }
gfCNCPoint3[24393] = {X 241.1102, Y 31.5690, Z -4.6667, A 0.000, B 0.000, C 0.000 }
gfCNCPoint3[24394] = {X 240.0470, Y 30.6432, Z -4.6667, A 0.000, B 0.000, C 0.000 }
gfCNCPoint3[24395] = {X 239.1072, Y 29.5925, Z -4.6667, A 0.000, B 0.000, C 0.000 }
gfCNCPoint3[24396] = {X 238.3052, Y 28.4330, Z -4.6667, A 0.000, B 0.000, C 0.000 }
gfCNCPoint3[24397] = {X 237.6537, Y 27.1829, Z -4.6667, A 0.000, B 0.000, C 0.000 }
gfCNCPoint3[24398] = {X 237.1626, Y 25.8614, Z -4.6667, A 0.000, B 0.000, C 0.000 }
gfCNCPoint3[24399] = {X 236.7424, Y 24.0500, Z -4.6667, A 0.000, B 0.000, C 0.000 }
gfCNCPoint3[24400] = {X 236.5283, Y 22.2028, Z -4.6667, A 0.000, B 0.000, C 0.000 }
gfCNCPoint3[24401] = {X 236.5230, Y 20.3432, Z -4.6667, A 0.000, B 0.000, C 0.000 }
gfCNCPoint3[24402] = {X 236.7264, Y 18.4948, Z -4.6667, A 0.000, B 0.000, C 0.000 }
gfCNCPoint3[24403] = {X 237.1362, Y 16.6809, Z -4.6667, A 0.000, B 0.000, C 0.000 }
gfCNCPoint3[24404] = {X 237.7066, Y 15.1053, Z -4.6667, A 0.000, B 0.000, C 0.000 }
gfCNCPoint3[24405] = {X 238.4936, Y 13.6258, Z -4.6667, A 0.000, B 0.000, C 0.000 }
gfCNCPoint3[24406] = {X 239.4814, Y 12.2722, Z -4.6667, A 0.000, B 0.000, C 0.000 }
gfCNCPoint3[24407] = {X 240.6503, Y 11.0715, Z -4.6667, A 0.000, B 0.000, C 0.000 }
gfCNCPoint3[24408] = {X 241.9770, Y 10.0477, Z -4.6667, A 0.000, B 0.000, C 0.000 }
gfCNCPoint3[24409] = {X 243.4348, Y 9.2213, Z -4.6667, A 0.000, B 0.000, C 0.000 }
gfCNCPoint3[24410] = {X 244.9946, Y 8.6088, Z -4.6667, A 0.000, B 0.000, C 0.000 }
gfCNCPoint3[24411] = {X 246.6252, Y 8.2226, Z -4.6667, A 0.000, B 0.000, C 0.000 }
gfCNCPoint3[24412] = {X 248.7221, Y 7.9511, Z -4.6667, A 0.000, B 0.000, C 0.000 }
gfCNCPoint3[24413] = {X 250.8350, Y 7.8706, Z -4.6667, A 0.000, B 0.000, C 0.000 }
gfCNCPoint3[24414] = {X 266.7633, Y 7.8706, Z -4.6667, A 0.000, B 0.000, C 0.000 }
gfCNCPoint3[24415] = {X 267.7185, Y 7.9853, Z -4.6667, A 0.000, B 0.000, C 0.000 }
gfCNCPoint3[24416] = {X 268.6247, Y 8.3085, Z -4.6667, A 0.000, B 0.000, C 0.000 }
gfCNCPoint3[24417] = {X 269.4369, Y 8.8242, Z -4.6667, A 0.000, B 0.000, C 0.000 }
gfCNCPoint3[24418] = {X 270.1149, Y 9.5067, Z -4.6667, A 0.000, B 0.000, C 0.000 }
gfCNCPoint3[24419] = {X 270.6252, Y 10.3222, Z -4.6667, A 0.000, B 0.000, C 0.000 }
gfCNCPoint3[24420] = {X 270.9425, Y 11.2305, Z -4.6667, A 0.000, B 0.000, C 0.000 }
gfCNCPoint3[24421] = {X 271.0510, Y 12.1864, Z -4.6667, A 0.000, B 0.000, C 0.000 }
gfCNCPoint3[24422] = {X 271.0508, Y 13.0225, Z -4.6667, A 0.000, B 0.000, C 0.000 }
gfCNCPoint3[24423] = {X 270.9425, Y 13.9404, Z -4.6667, A 0.000, B 0.000, C 0.000 }
gfCNCPoint3[24424] = {X 270.6413, Y 14.8143, Z -4.6667, A 0.000, B 0.000, C 0.000 }
gfCNCPoint3[24425] = {X 270.1612, Y 15.6041, Z -4.6667, A 0.000, B 0.000, C 0.000 }
gfCNCPoint3[24426] = {X 269.5240, Y 16.2737, Z -4.6667, A 0.000, B 0.000, C 0.000 }
gfCNCPoint3[24427] = {X 269.5239, Y 28.5936, Z -4.6667, A 0.000, B 0.000, C 0.000 }
gfCNCPoint3[24428] = {X 273.5239, Y 28.5936, Z -4.6667, A 0.000, B 0.000, C 0.000 }
gfCNCPoint3[24429] = {X 269.4439, Y 28.5936, Z -4.6667, A 0.000, B 0.000, C 0.000 }
gfCNCPoint3[24430] = {X 269.4439, Y 40.9516, Z -4.6667, A 0.000, B 0.000, C 0.000 }
gfCNCPoint3[24431] = {X 269.4862, Y 40.9860, Z -4.6667, A 0.000, B 0.000, C 0.000 }
gfCNCPoint3[24432] = {X 270.1066, Y 41.6431, Z -4.6667, A 0.000, B 0.000, C 0.000 }
gfCNCPoint3[24433] = {X 270.5737, Y 42.4167, Z -4.6667, A 0.000, B 0.000, C 0.000 }
gfCNCPoint3[24434] = {X 270.8662, Y 43.2717, Z -4.6667, A 0.000, B 0.000, C 0.000 }
gfCNCPoint3[24435] = {X 270.9708, Y 44.1693, Z -4.6667, A 0.000, B 0.000, C 0.000 }
gfCNCPoint3[24436] = {X 270.9710, Y 45.0000, Z -4.6667, A 0.000, B 0.000, C 0.000 }
gfCNCPoint3[24437] = {X 270.8647, Y 45.9435, Z -4.6667, A 0.000, B 0.000, C 0.000 }
gfCNCPoint3[24438] = {X 270.5511, Y 46.8397, Z -4.6667, A 0.000, B 0.000, C 0.000 }
gfCNCPoint3[24439] = {X 270.0460, Y 47.6436, Z -4.6667, A 0.000, B 0.000, C 0.000 }
gfCNCPoint3[24440] = {X 269.3746, Y 48.3150, Z -4.6667, A 0.000, B 0.000, C 0.000 }
gfCNCPoint3[24441] = {X 268.5707, Y 48.8201, Z -4.6667, A 0.000, B 0.000, C 0.000 }
gfCNCPoint3[24442] = {X 267.6745, Y 49.1337, Z -4.6667, A 0.000, B 0.000, C 0.000 }
gfCNCPoint3[24443] = {X 266.7310, Y 49.2400, Z -4.6667, A 0.000, B 0.000, C 0.000 }
gfCNCPoint3[24444] = {X 260.2876, Y 49.2400, Z -4.6667, A 0.000, B 0.000, C 0.000 }
gfCNCPoint3[24445] = {X 259.3487, Y 49.1347, Z -4.6667, A 0.000, B 0.000, C 0.000 }
gfCNCPoint3[24446] = {X 258.4564, Y 48.8242, Z -4.6667, A 0.000, B 0.000, C 0.000 }
gfCNCPoint3[24447] = {X 257.6550, Y 48.3238, Z -4.6667, A 0.000, B 0.000, C 0.000 }
gfCNCPoint3[24448] = {X 256.9844, Y 47.6583, Z -4.6667, A 0.000, B 0.000, C 0.000 }
gfCNCPoint3[24449] = {X 256.4777, Y 46.8609, Z -4.6667, A 0.000, B 0.000, C 0.000 }
gfCNCPoint3[24450] = {X 256.1603, Y 45.9711, Z -4.6667, A 0.000, B 0.000, C 0.000 }
gfCNCPoint3[24451] = {X 256.0477, Y 45.0330, Z -4.6667, A 0.000, B 0.000, C 0.000 }
gfCNCPoint3[24452] = {X 256.0480, Y 44.1505, Z -4.6667, A 0.000, B 0.000, C 0.000 }
gfCNCPoint3[24453] = {X 256.1585, Y 43.2454, Z -4.6667, A 0.000, B 0.000, C 0.000 }
gfCNCPoint3[24454] = {X 256.4599, Y 42.3850, Z -4.6667, A 0.000, B 0.000, C 0.000 }
gfCNCPoint3[24455] = {X 256.9383, Y 41.6088, Z -4.6667, A 0.000, B 0.000, C 0.000 }
gfCNCPoint3[24456] = {X 257.5715, Y 40.9529, Z -4.6667, A 0.000, B 0.000, C 0.000 }
gfCNCPoint3[24457] = {X 257.5715, Y 34.3938, Z -4.6667, A 0.000, B 0.000, C 0.000 }
gfCNCPoint3[24458] = {X 254.7188, Y 34.3938, Z -4.6667, A 0.000, B 0.000, C 0.000 }
gfCNCPoint3[24459] = {X 250.3970, Y 42.8124, Z -4.6667, A 0.000, B 0.000, C 0.000 }
gfCNCPoint3[24460] = {X 250.5710, Y 43.4830, Z -4.6667, A 0.000, B 0.000, C 0.000 }
gfCNCPoint3[24461] = {X 250.6334, Y 44.1730, Z -4.6667, A 0.000, B 0.000, C 0.000 }
gfCNCPoint3[24462] = {X 250.6336, Y 45.0000, Z -4.6667, A 0.000, B 0.000, C 0.000 }
gfCNCPoint3[24463] = {X 250.5273, Y 45.9435, Z -4.6667, A 0.000, B 0.000, C 0.000 }
gfCNCPoint3[24464] = {X 250.2137, Y 46.8397, Z -4.6667, A 0.000, B 0.000, C 0.000 }
gfCNCPoint3[24465] = {X 249.7085, Y 47.6436, Z -4.6667, A 0.000, B 0.000, C 0.000 }
gfCNCPoint3[24466] = {X 249.0372, Y 48.3150, Z -4.6667, A 0.000, B 0.000, C 0.000 }
gfCNCPoint3[24467] = {X 248.2332, Y 48.8201, Z -4.6667, A 0.000, B 0.000, C 0.000 }
gfCNCPoint3[24468] = {X 247.3370, Y 49.1337, Z -4.6667, A 0.000, B 0.000, C 0.000 }
gfCNCPoint3[24469] = {X 246.3936, Y 49.2400, Z -4.6667, A 0.000, B 0.000, C 0.000 }
gfCNCPoint3[24470] = {X 239.8075, Y 49.2400, Z -4.6667, A 0.000, B 0.000, C 0.000 }
gfCNCPoint3[24471] = {X 238.8640, Y 49.1337, Z -4.6667, A 0.000, B 0.000, C 0.000 }
gfCNCPoint3[24472] = {X 237.9679, Y 48.8201, Z -4.6667, A 0.000, B 0.000, C 0.000 }
gfCNCPoint3[24473] = {X 237.1639, Y 48.3150, Z -4.6667, A 0.000, B 0.000, C 0.000 }
gfCNCPoint3[24474] = {X 236.4926, Y 47.6436, Z -4.6667, A 0.000, B 0.000, C 0.000 }
gfCNCPoint3[24475] = {X 235.9874, Y 46.8397, Z -4.6667, A 0.000, B 0.000, C 0.000 }
gfCNCPoint3[24476] = {X 235.6738, Y 45.9436, Z -4.6667, A 0.000, B 0.000, C 0.000 }
gfCNCPoint3[24477] = {X 235.5675, Y 45.0001, Z -4.6667, A 0.000, B 0.000, C 0.000 }
gfCNCPoint3[24478] = {X 235.5679, Y 44.1505, Z -4.6667, A 0.000, B 0.000, C 0.000 }
gfCNCPoint3[24479] = {X 235.6649, Y 43.3054, Z -4.6667, A 0.000, B 0.000, C 0.000 }
gfCNCPoint3[24480] = {X 235.9285, Y 42.4967, Z -4.6667, A 0.000, B 0.000, C 0.000 }
gfCNCPoint3[24481] = {X 236.3483, Y 41.7570, Z -4.6667, A 0.000, B 0.000, C 0.000 }
gfCNCPoint3[24482] = {X 236.9073, Y 41.1159, Z -4.6667, A 0.000, B 0.000, C 0.000 }
gfCNCPoint3[24483] = {X 237.5830, Y 40.5992, Z -4.6667, A 0.000, B 0.000, C 0.000 }
gfCNCPoint3[24484] = {X 238.3482, Y 40.2278, Z -4.6667, A 0.000, B 0.000, C 0.000 }
gfCNCPoint3[24485] = {X 242.3860, Y 32.3243, Z -4.6667, A 0.000, B 0.000, C 0.000 }
gfCNCPoint3[24486] = {X 241.2090, Y 31.5437, Z -4.6667, A 0.000, B 0.000, C 0.000 }
gfCNCPoint3[24487] = {X 240.1392, Y 30.6216, Z -4.6667, A 0.000, B 0.000, C 0.000 }
gfCNCPoint3[24488] = {X 239.1934, Y 29.5726, Z -4.6667, A 0.000, B 0.000, C 0.000 }
gfCNCPoint3[24489] = {X 238.3868, Y 28.4133, Z -4.6667, A 0.000, B 0.000, C 0.000 }
gfCNCPoint3[24490] = {X 237.7319, Y 27.1619, Z -4.6667, A 0.000, B 0.000, C 0.000 }
gfCNCPoint3[24491] = {X 237.2392, Y 25.8383, Z -4.6667, A 0.000, B 0.000, C 0.000 }
gfCNCPoint3[24492] = {X 236.8211, Y 24.0357, Z -4.6667, A 0.000, B 0.000, C 0.000 }
gfCNCPoint3[24493] = {X 236.6081, Y 22.1976, Z -4.6667, A 0.000, B 0.000, C 0.000 }
gfCNCPoint3[24494] = {X 236.6029, Y 20.3471, Z -4.6667, A 0.000, B 0.000, C 0.000 }
gfCNCPoint3[24495] = {X 236.8054, Y 18.5078, Z -4.6667, A 0.000, B 0.000, C 0.000 }
gfCNCPoint3[24496] = {X 237.2131, Y 16.7029, Z -4.6667, A 0.000, B 0.000, C 0.000 }
gfCNCPoint3[24497] = {X 237.7797, Y 15.1378, Z -4.6667, A 0.000, B 0.000, C 0.000 }
gfCNCPoint3[24498] = {X 238.5614, Y 13.6682, Z -4.6667, A 0.000, B 0.000, C 0.000 }
gfCNCPoint3[24499] = {X 239.5426, Y 12.3237, Z -4.6667, A 0.000, B 0.000, C 0.000 }
gfCNCPoint3[24500] = {X 240.7037, Y 11.1311, Z -4.6667, A 0.000, B 0.000, C 0.000 }
gfCNCPoint3[24501] = {X 242.0215, Y 10.1142, Z -4.6667, A 0.000, B 0.000, C 0.000 }
gfCNCPoint3[24502] = {X 243.4695, Y 9.2934, Z -4.6667, A 0.000, B 0.000, C 0.000 }
gfCNCPoint3[24503] = {X 245.0189, Y 8.6851, Z -4.6667, A 0.000, B 0.000, C 0.000 }
gfCNCPoint3[24504] = {X 246.6386, Y 8.3015, Z -4.6667, A 0.000, B 0.000, C 0.000 }
gfCNCPoint3[24505] = {X 248.7287, Y 8.0308, Z -4.6667, A 0.000, B 0.000, C 0.000 }
gfCNCPoint3[24506] = {X 250.8346, Y 7.9506, Z -4.6667, A 0.000, B 0.000, C 0.000 }
gfCNCPoint3[24507] = {X 266.7627, Y 7.9506, Z -4.6667, A 0.000, B 0.000, C 0.000 }
gfCNCPoint3[24508] = {X 267.7002, Y 8.0632, Z -4.6667, A 0.000, B 0.000, C 0.000 }
gfCNCPoint3[24509] = {X 268.5896, Y 8.3804, Z -4.6667, A 0.000, B 0.000, C 0.000 }
gfCNCPoint3[24510] = {X 269.3868, Y 8.8865, Z -4.6667, A 0.000, B 0.000, C 0.000 }
gfCNCPoint3[24511] = {X 270.0523, Y 9.5564, Z -4.6667, A 0.000, B 0.000, C 0.000 }
gfCNCPoint3[24512] = {X 270.5531, Y 10.3568, Z -4.6667, A 0.000, B 0.000, C 0.000 }
gfCNCPoint3[24513] = {X 270.8645, Y 11.2483, Z -4.6667, A 0.000, B 0.000, C 0.000 }
gfCNCPoint3[24514] = {X 270.9710, Y 12.1865, Z -4.6667, A 0.000, B 0.000, C 0.000 }
gfCNCPoint3[24515] = {X 270.9708, Y 13.0217, Z -4.6667, A 0.000, B 0.000, C 0.000 }
gfCNCPoint3[24516] = {X 270.8624, Y 13.9316, Z -4.6667, A 0.000, B 0.000, C 0.000 }
gfCNCPoint3[24517] = {X 270.5610, Y 14.7970, Z -4.6667, A 0.000, B 0.000, C 0.000 }
gfCNCPoint3[24518] = {X 270.0808, Y 15.5774, Z -4.6667, A 0.000, B 0.000, C 0.000 }
gfCNCPoint3[24519] = {X 269.4440, Y 16.2364, Z -4.6667, A 0.000, B 0.000, C 0.000 }
gfCNCPoint3[24520] = {X 269.4439, Y 28.5936, Z -4.6667, A 0.000, B 0.000, C 0.000 }
gfCNCPoint3[24521] = {X 273.4439, Y 28.5936, Z -4.6667, A 0.000, B 0.000, C 0.000 }
gfCNCPoint3[24522] = {X 269.3639, Y 28.5936, Z -4.6667, A 0.000, B 0.000, C 0.000 }
gfCNCPoint3[24523] = {X 269.3639, Y 40.9896, Z -4.6667, A 0.000, B 0.000, C 0.000 }
gfCNCPoint3[24524] = {X 269.4350, Y 41.0474, Z -4.6667, A 0.000, B 0.000, C 0.000 }
gfCNCPoint3[24525] = {X 270.0434, Y 41.6921, Z -4.6667, A 0.000, B 0.000, C 0.000 }
gfCNCPoint3[24526] = {X 270.5014, Y 42.4509, Z -4.6667, A 0.000, B 0.000, C 0.000 }
gfCNCPoint3[24527] = {X 270.7882, Y 43.2896, Z -4.6667, A 0.000, B 0.000, C 0.000 }
gfCNCPoint3[24528] = {X 270.8909, Y 44.1700, Z -4.6667, A 0.000, B 0.000, C 0.000 }
gfCNCPoint3[24529] = {X 270.8910, Y 45.0000, Z -4.6667, A 0.000, B 0.000, C 0.000 }
gfCNCPoint3[24530] = {X 270.7867, Y 45.9257, Z -4.6667, A 0.000, B 0.000, C 0.000 }
gfCNCPoint3[24531] = {X 270.4791, Y 46.8050, Z -4.6667, A 0.000, B 0.000, C 0.000 }
gfCNCPoint3[24532] = {X 269.9835, Y 47.5937, Z -4.6667, A 0.000, B 0.000, C 0.000 }
gfCNCPoint3[24533] = {X 269.3247, Y 48.2524, Z -4.6667, A 0.000, B 0.000, C 0.000 }
gfCNCPoint3[24534] = {X 268.5360, Y 48.7480, Z -4.6667, A 0.000, B 0.000, C 0.000 }
gfCNCPoint3[24535] = {X 267.6567, Y 49.0557, Z -4.6667, A 0.000, B 0.000, C 0.000 }
gfCNCPoint3[24536] = {X 266.7310, Y 49.1600, Z -4.6667, A 0.000, B 0.000, C 0.000 }
gfCNCPoint3[24537] = {X 260.2876, Y 49.1600, Z -4.6667, A 0.000, B 0.000, C 0.000 }
gfCNCPoint3[24538] = {X 259.3664, Y 49.0567, Z -4.6667, A 0.000, B 0.000, C 0.000 }
gfCNCPoint3[24539] = {X 258.4910, Y 48.7520, Z -4.6667, A 0.000, B 0.000, C 0.000 }
gfCNCPoint3[24540] = {X 257.7047, Y 48.2611, Z -4.6667, A 0.000, B 0.000, C 0.000 }
gfCNCPoint3[24541] = {X 257.0467, Y 47.6082, Z -4.6667, A 0.000, B 0.000, C 0.000 }
gfCNCPoint3[24542] = {X 256.5496, Y 46.8258, Z -4.6667, A 0.000, B 0.000, C 0.000 }
gfCNCPoint3[24543] = {X 256.2381, Y 45.9527, Z -4.6667, A 0.000, B 0.000, C 0.000 }
gfCNCPoint3[24544] = {X 256.1277, Y 45.0324, Z -4.6667, A 0.000, B 0.000, C 0.000 }
gfCNCPoint3[24545] = {X 256.1280, Y 44.1516, Z -4.6667, A 0.000, B 0.000, C 0.000 }
gfCNCPoint3[24546] = {X 256.2385, Y 43.2545, Z -4.6667, A 0.000, B 0.000, C 0.000 }
gfCNCPoint3[24547] = {X 256.5401, Y 42.4026, Z -4.6667, A 0.000, B 0.000, C 0.000 }
gfCNCPoint3[24548] = {X 257.0187, Y 41.6358, Z -4.6667, A 0.000, B 0.000, C 0.000 }
gfCNCPoint3[24549] = {X 257.6515, Y 40.9906, Z -4.6667, A 0.000, B 0.000, C 0.000 }
gfCNCPoint3[24550] = {X 257.6515, Y 34.3138, Z -4.6667, A 0.000, B 0.000, C 0.000 }
gfCNCPoint3[24551] = {X 254.6700, Y 34.3138, Z -4.6667, A 0.000, B 0.000, C 0.000 }
gfCNCPoint3[24552] = {X 250.3101, Y 42.8066, Z -4.6667, A 0.000, B 0.000, C 0.000 }
gfCNCPoint3[24553] = {X 250.4892, Y 43.4799, Z -4.6667, A 0.000, B 0.000, C 0.000 }
gfCNCPoint3[24554] = {X 250.5534, Y 44.1736, Z -4.6667, A 0.000, B 0.000, C 0.000 }
gfCNCPoint3[24555] = {X 250.5536, Y 45.0000, Z -4.6667, A 0.000, B 0.000, C 0.000 }
gfCNCPoint3[24556] = {X 250.4493, Y 45.9257, Z -4.6667, A 0.000, B 0.000, C 0.000 }
gfCNCPoint3[24557] = {X 250.1416, Y 46.8050, Z -4.6667, A 0.000, B 0.000, C 0.000 }
gfCNCPoint3[24558] = {X 249.6460, Y 47.5937, Z -4.6667, A 0.000, B 0.000, C 0.000 }
gfCNCPoint3[24559] = {X 248.9873, Y 48.2524, Z -4.6667, A 0.000, B 0.000, C 0.000 }
gfCNCPoint3[24560] = {X 248.1985, Y 48.7480, Z -4.6667, A 0.000, B 0.000, C 0.000 }
gfCNCPoint3[24561] = {X 247.3192, Y 49.0557, Z -4.6667, A 0.000, B 0.000, C 0.000 }
gfCNCPoint3[24562] = {X 246.3936, Y 49.1600, Z -4.6667, A 0.000, B 0.000, C 0.000 }
gfCNCPoint3[24563] = {X 239.8075, Y 49.1600, Z -4.6667, A 0.000, B 0.000, C 0.000 }
gfCNCPoint3[24564] = {X 238.8818, Y 49.0557, Z -4.6667, A 0.000, B 0.000, C 0.000 }
gfCNCPoint3[24565] = {X 238.0026, Y 48.7480, Z -4.6667, A 0.000, B 0.000, C 0.000 }
gfCNCPoint3[24566] = {X 237.2138, Y 48.2524, Z -4.6667, A 0.000, B 0.000, C 0.000 }
gfCNCPoint3[24567] = {X 236.5551, Y 47.5937, Z -4.6667, A 0.000, B 0.000, C 0.000 }
gfCNCPoint3[24568] = {X 236.0595, Y 46.8050, Z -4.6667, A 0.000, B 0.000, C 0.000 }
gfCNCPoint3[24569] = {X 235.7518, Y 45.9257, Z -4.6667, A 0.000, B 0.000, C 0.000 }
gfCNCPoint3[24570] = {X 235.6475, Y 45.0000, Z -4.6667, A 0.000, B 0.000, C 0.000 }
gfCNCPoint3[24571] = {X 235.6479, Y 44.1516, Z -4.6667, A 0.000, B 0.000, C 0.000 }
gfCNCPoint3[24572] = {X 235.7441, Y 43.3174, Z -4.6667, A 0.000, B 0.000, C 0.000 }
gfCNCPoint3[24573] = {X 236.0059, Y 42.5195, Z -4.6667, A 0.000, B 0.000, C 0.000 }
gfCNCPoint3[24574] = {X 236.4226, Y 41.7905, Z -4.6667, A 0.000, B 0.000, C 0.000 }
gfCNCPoint3[24575] = {X 236.9772, Y 41.1600, Z -4.6667, A 0.000, B 0.000, C 0.000 }
gfCNCPoint3[24576] = {X 237.6471, Y 40.6537, Z -4.6667, A 0.000, B 0.000, C 0.000 }
gfCNCPoint3[24577] = {X 238.4051, Y 40.2923, Z -4.6667, A 0.000, B 0.000, C 0.000 }
gfCNCPoint3[24578] = {X 242.4920, Y 32.2927, Z -4.6667, A 0.000, B 0.000, C 0.000 }
gfCNCPoint3[24579] = {X 241.3079, Y 31.5181, Z -4.6667, A 0.000, B 0.000, C 0.000 }
gfCNCPoint3[24580] = {X 240.2314, Y 30.5998, Z -4.6667, A 0.000, B 0.000, C 0.000 }
gfCNCPoint3[24581] = {X 239.2798, Y 29.5526, Z -4.6667, A 0.000, B 0.000, C 0.000 }
gfCNCPoint3[24582] = {X 238.4684, Y 28.3935, Z -4.6667, A 0.000, B 0.000, C 0.000 }
gfCNCPoint3[24583] = {X 237.8101, Y 27.1409, Z -4.6667, A 0.000, B 0.000, C 0.000 }
gfCNCPoint3[24584] = {X 237.3158, Y 25.8152, Z -4.6667, A 0.000, B 0.000, C 0.000 }
gfCNCPoint3[24585] = {X 236.8999, Y 24.0214, Z -4.6667, A 0.000, B 0.000, C 0.000 }
gfCNCPoint3[24586] = {X 236.6880, Y 22.1924, Z -4.6667, A 0.000, B 0.000, C 0.000 }
gfCNCPoint3[24587] = {X 236.6828, Y 20.3511, Z -4.6667, A 0.000, B 0.000, C 0.000 }
gfCNCPoint3[24588] = {X 236.8843, Y 18.5209, Z -4.6667, A 0.000, B 0.000, C 0.000 }
gfCNCPoint3[24589] = {X 237.2900, Y 16.7248, Z -4.6667, A 0.000, B 0.000, C 0.000 }
gfCNCPoint3[24590] = {X 237.8528, Y 15.1703, Z -4.6667, A 0.000, B 0.000, C 0.000 }
gfCNCPoint3[24591] = {X 238.6292, Y 13.7107, Z -4.6667, A 0.000, B 0.000, C 0.000 }
gfCNCPoint3[24592] = {X 239.6038, Y 12.3752, Z -4.6667, A 0.000, B 0.000, C 0.000 }
gfCNCPoint3[24593] = {X 240.7571, Y 11.1906, Z -4.6667, A 0.000, B 0.000, C 0.000 }
gfCNCPoint3[24594] = {X 242.0660, Y 10.1806, Z -4.6667, A 0.000, B 0.000, C 0.000 }
gfCNCPoint3[24595] = {X 243.5043, Y 9.3654, Z -4.6667, A 0.000, B 0.000, C 0.000 }
gfCNCPoint3[24596] = {X 245.0432, Y 8.7613, Z -4.6667, A 0.000, B 0.000, C 0.000 }
gfCNCPoint3[24597] = {X 246.6520, Y 8.3803, Z -4.6667, A 0.000, B 0.000, C 0.000 }
gfCNCPoint3[24598] = {X 248.7352, Y 8.1106, Z -4.6667, A 0.000, B 0.000, C 0.000 }
gfCNCPoint3[24599] = {X 250.8343, Y 8.0306, Z -4.6667, A 0.000, B 0.000, C 0.000 }
gfCNCPoint3[24600] = {X 266.7621, Y 8.0306, Z -4.6667, A 0.000, B 0.000, C 0.000 }
gfCNCPoint3[24601] = {X 267.6819, Y 8.1411, Z -4.6667, A 0.000, B 0.000, C 0.000 }
gfCNCPoint3[24602] = {X 268.5545, Y 8.4523, Z -4.6667, A 0.000, B 0.000, C 0.000 }
gfCNCPoint3[24603] = {X 269.3366, Y 8.9489, Z -4.6667, A 0.000, B 0.000, C 0.000 }
gfCNCPoint3[24604] = {X 269.9896, Y 9.6061, Z -4.6667, A 0.000, B 0.000, C 0.000 }
gfCNCPoint3[24605] = {X 270.4810, Y 10.3915, Z -4.6667, A 0.000, B 0.000, C 0.000 }
gfCNCPoint3[24606] = {X 270.7865, Y 11.2661, Z -4.6667, A 0.000, B 0.000, C 0.000 }
gfCNCPoint3[24607] = {X 270.8910, Y 12.1866, Z -4.6667, A 0.000, B 0.000, C 0.000 }
gfCNCPoint3[24608] = {X 270.8908, Y 13.0208, Z -4.6667, A 0.000, B 0.000, C 0.000 }
gfCNCPoint3[24609] = {X 270.7824, Y 13.9227, Z -4.6667, A 0.000, B 0.000, C 0.000 }
gfCNCPoint3[24610] = {X 270.4807, Y 14.7795, Z -4.6667, A 0.000, B 0.000, C 0.000 }
gfCNCPoint3[24611] = {X 270.0003, Y 15.5504, Z -4.6667, A 0.000, B 0.000, C 0.000 }
gfCNCPoint3[24612] = {X 269.3640, Y 16.1987, Z -4.6667, A 0.000, B 0.000, C 0.000 }
gfCNCPoint3[24613] = {X 269.3639, Y 28.5936, Z -4.6667, A 0.000, B 0.000, C 0.000 }
gfCNCPoint3[24614] = {X 273.3639, Y 28.5936, Z -4.6667, A 0.000, B 0.000, C 0.000 }
gfCNCPoint3[24615] = {X 269.2839, Y 28.5936, Z -4.6667, A 0.000, B 0.000, C 0.000 }
gfCNCPoint3[24616] = {X 269.2839, Y 41.0277, Z -4.6667, A 0.000, B 0.000, C 0.000 }
gfCNCPoint3[24617] = {X 269.3838, Y 41.1089, Z -4.6667, A 0.000, B 0.000, C 0.000 }
gfCNCPoint3[24618] = {X 269.9801, Y 41.7411, Z -4.6667, A 0.000, B 0.000, C 0.000 }
gfCNCPoint3[24619] = {X 270.4291, Y 42.4852, Z -4.6667, A 0.000, B 0.000, C 0.000 }
gfCNCPoint3[24620] = {X 270.7102, Y 43.3075, Z -4.6667, A 0.000, B 0.000, C 0.000 }
gfCNCPoint3[24621] = {X 270.8109, Y 44.1708, Z -4.6667, A 0.000, B 0.000, C 0.000 }
gfCNCPoint3[24622] = {X 270.8110, Y 45.0000, Z -4.6667, A 0.000, B 0.000, C 0.000 }
gfCNCPoint3[24623] = {X 270.7087, Y 45.9079, Z -4.6667, A 0.000, B 0.000, C 0.000 }
gfCNCPoint3[24624] = {X 270.4070, Y 46.7702, Z -4.6667, A 0.000, B 0.000, C 0.000 }
gfCNCPoint3[24625] = {X 269.9209, Y 47.5438, Z -4.6667, A 0.000, B 0.000, C 0.000 }
gfCNCPoint3[24626] = {X 269.2749, Y 48.1899, Z -4.6667, A 0.000, B 0.000, C 0.000 }
gfCNCPoint3[24627] = {X 268.5013, Y 48.6760, Z -4.6667, A 0.000, B 0.000, C 0.000 }
gfCNCPoint3[24628] = {X 267.6389, Y 48.9777, Z -4.6667, A 0.000, B 0.000, C 0.000 }
gfCNCPoint3[24629] = {X 266.7310, Y 49.0800, Z -4.6667, A 0.000, B 0.000, C 0.000 }
gfCNCPoint3[24630] = {X 260.2876, Y 49.0800, Z -4.6667, A 0.000, B 0.000, C 0.000 }
gfCNCPoint3[24631] = {X 259.3841, Y 48.9787, Z -4.6667, A 0.000, B 0.000, C 0.000 }
gfCNCPoint3[24632] = {X 258.5255, Y 48.6799, Z -4.6667, A 0.000, B 0.000, C 0.000 }
gfCNCPoint3[24633] = {X 257.7544, Y 48.1983, Z -4.6667, A 0.000, B 0.000, C 0.000 }
gfCNCPoint3[24634] = {X 257.1090, Y 47.5580, Z -4.6667, A 0.000, B 0.000, C 0.000 }
gfCNCPoint3[24635] = {X 256.6215, Y 46.7907, Z -4.6667, A 0.000, B 0.000, C 0.000 }
gfCNCPoint3[24636] = {X 256.3160, Y 45.9344, Z -4.6667, A 0.000, B 0.000, C 0.000 }
gfCNCPoint3[24637] = {X 256.2077, Y 45.0318, Z -4.6667, A 0.000, B 0.000, C 0.000 }
gfCNCPoint3[24638] = {X 256.2080, Y 44.1527, Z -4.6667, A 0.000, B 0.000, C 0.000 }
gfCNCPoint3[24639] = {X 256.3185, Y 43.2637, Z -4.6667, A 0.000, B 0.000, C 0.000 }
gfCNCPoint3[24640] = {X 256.6204, Y 42.4203, Z -4.6667, A 0.000, B 0.000, C 0.000 }
gfCNCPoint3[24641] = {X 257.0991, Y 41.6631, Z -4.6667, A 0.000, B 0.000, C 0.000 }
gfCNCPoint3[24642] = {X 257.7315, Y 41.0287, Z -4.6667, A 0.000, B 0.000, C 0.000 }
gfCNCPoint3[24643] = {X 257.7315, Y 34.2338, Z -4.6667, A 0.000, B 0.000, C 0.000 }
gfCNCPoint3[24644] = {X 254.6211, Y 34.2338, Z -4.6667, A 0.000, B 0.000, C 0.000 }
gfCNCPoint3[24645] = {X 250.2230, Y 42.8011, Z -4.6667, A 0.000, B 0.000, C 0.000 }
gfCNCPoint3[24646] = {X 250.4074, Y 43.4769, Z -4.6667, A 0.000, B 0.000, C 0.000 }
gfCNCPoint3[24647] = {X 250.4734, Y 44.1743, Z -4.6667, A 0.000, B 0.000, C 0.000 }
gfCNCPoint3[24648] = {X 250.4736, Y 45.0000, Z -4.6667, A 0.000, B 0.000, C 0.000 }
gfCNCPoint3[24649] = {X 250.3713, Y 45.9079, Z -4.6667, A 0.000, B 0.000, C 0.000 }
gfCNCPoint3[24650] = {X 250.0695, Y 46.7702, Z -4.6667, A 0.000, B 0.000, C 0.000 }
gfCNCPoint3[24651] = {X 249.5834, Y 47.5438, Z -4.6667, A 0.000, B 0.000, C 0.000 }
gfCNCPoint3[24652] = {X 248.9374, Y 48.1899, Z -4.6667, A 0.000, B 0.000, C 0.000 }
gfCNCPoint3[24653] = {X 248.1638, Y 48.6760, Z -4.6667, A 0.000, B 0.000, C 0.000 }
gfCNCPoint3[24654] = {X 247.3014, Y 48.9777, Z -4.6667, A 0.000, B 0.000, C 0.000 }
gfCNCPoint3[24655] = {X 246.3936, Y 49.0800, Z -4.6667, A 0.000, B 0.000, C 0.000 }
gfCNCPoint3[24656] = {X 239.8075, Y 49.0800, Z -4.6667, A 0.000, B 0.000, C 0.000 }
gfCNCPoint3[24657] = {X 238.8996, Y 48.9777, Z -4.6667, A 0.000, B 0.000, C 0.000 }
gfCNCPoint3[24658] = {X 238.0373, Y 48.6760, Z -4.6667, A 0.000, B 0.000, C 0.000 }
gfCNCPoint3[24659] = {X 237.2637, Y 48.1899, Z -4.6667, A 0.000, B 0.000, C 0.000 }
gfCNCPoint3[24660] = {X 236.6176, Y 47.5438, Z -4.6667, A 0.000, B 0.000, C 0.000 }
gfCNCPoint3[24661] = {X 236.1315, Y 46.7702, Z -4.6667, A 0.000, B 0.000, C 0.000 }
gfCNCPoint3[24662] = {X 235.8298, Y 45.9079, Z -4.6667, A 0.000, B 0.000, C 0.000 }
gfCNCPoint3[24663] = {X 235.7275, Y 45.0000, Z -4.6667, A 0.000, B 0.000, C 0.000 }
gfCNCPoint3[24664] = {X 235.7279, Y 44.1527, Z -4.6667, A 0.000, B 0.000, C 0.000 }
gfCNCPoint3[24665] = {X 235.8234, Y 43.3294, Z -4.6667, A 0.000, B 0.000, C 0.000 }
gfCNCPoint3[24666] = {X 236.0833, Y 42.5424, Z -4.6667, A 0.000, B 0.000, C 0.000 }
gfCNCPoint3[24667] = {X 236.4969, Y 41.8242, Z -4.6667, A 0.000, B 0.000, C 0.000 }
gfCNCPoint3[24668] = {X 237.0471, Y 41.2044, Z -4.6667, A 0.000, B 0.000, C 0.000 }
gfCNCPoint3[24669] = {X 237.7112, Y 40.7085, Z -4.6667, A 0.000, B 0.000, C 0.000 }
gfCNCPoint3[24670] = {X 238.4618, Y 40.3571, Z -4.6667, A 0.000, B 0.000, C 0.000 }
gfCNCPoint3[24671] = {X 242.5982, Y 32.2607, Z -4.6667, A 0.000, B 0.000, C 0.000 }
gfCNCPoint3[24672] = {X 241.4070, Y 31.4921, Z -4.6667, A 0.000, B 0.000, C 0.000 }
gfCNCPoint3[24673] = {X 240.3238, Y 30.5778, Z -4.6667, A 0.000, B 0.000, C 0.000 }
gfCNCPoint3[24674] = {X 239.3662, Y 29.5325, Z -4.6667, A 0.000, B 0.000, C 0.000 }
gfCNCPoint3[24675] = {X 238.5500, Y 28.3736, Z -4.6667, A 0.000, B 0.000, C 0.000 }
gfCNCPoint3[24676] = {X 237.8884, Y 27.1199, Z -4.6667, A 0.000, B 0.000, C 0.000 }
gfCNCPoint3[24677] = {X 237.3923, Y 25.7920, Z -4.6667, A 0.000, B 0.000, C 0.000 }
gfCNCPoint3[24678] = {X 236.9786, Y 24.0072, Z -4.6667, A 0.000, B 0.000, C 0.000 }
gfCNCPoint3[24679] = {X 236.7678, Y 22.1872, Z -4.6667, A 0.000, B 0.000, C 0.000 }
gfCNCPoint3[24680] = {X 236.7627, Y 20.3551, Z -4.6667, A 0.000, B 0.000, C 0.000 }
gfCNCPoint3[24681] = {X 236.9632, Y 18.5339, Z -4.6667, A 0.000, B 0.000, C 0.000 }
gfCNCPoint3[24682] = {X 237.3670, Y 16.7468, Z -4.6667, A 0.000, B 0.000, C 0.000 }
gfCNCPoint3[24683] = {X 237.9258, Y 15.2028, Z -4.6667, A 0.000, B 0.000, C 0.000 }
gfCNCPoint3[24684] = {X 238.6970, Y 13.7531, Z -4.6667, A 0.000, B 0.000, C 0.000 }
gfCNCPoint3[24685] = {X 239.6650, Y 12.4268, Z -4.6667, A 0.000, B 0.000, C 0.000 }
gfCNCPoint3[24686] = {X 240.8105, Y 11.2502, Z -4.6667, A 0.000, B 0.000, C 0.000 }
gfCNCPoint3[24687] = {X 242.1105, Y 10.2471, Z -4.6667, A 0.000, B 0.000, C 0.000 }
gfCNCPoint3[24688] = {X 243.5390, Y 9.4375, Z -4.6667, A 0.000, B 0.000, C 0.000 }
gfCNCPoint3[24689] = {X 245.0675, Y 8.8375, Z -4.6667, A 0.000, B 0.000, C 0.000 }
gfCNCPoint3[24690] = {X 246.6653, Y 8.4592, Z -4.6667, A 0.000, B 0.000, C 0.000 }
gfCNCPoint3[24691] = {X 248.7418, Y 8.1903, Z -4.6667, A 0.000, B 0.000, C 0.000 }
gfCNCPoint3[24692] = {X 250.8340, Y 8.1106, Z -4.6667, A 0.000, B 0.000, C 0.000 }
gfCNCPoint3[24693] = {X 266.7614, Y 8.1106, Z -4.6667, A 0.000, B 0.000, C 0.000 }
gfCNCPoint3[24694] = {X 267.6636, Y 8.2190, Z -4.6667, A 0.000, B 0.000, C 0.000 }
gfCNCPoint3[24695] = {X 268.5194, Y 8.5242, Z -4.6667, A 0.000, B 0.000, C 0.000 }
gfCNCPoint3[24696] = {X 269.2865, Y 9.0112, Z -4.6667, A 0.000, B 0.000, C 0.000 }
gfCNCPoint3[24697] = {X 269.9269, Y 9.6558, Z -4.6667, A 0.000, B 0.000, C 0.000 }
gfCNCPoint3[24698] = {X 270.4089, Y 10.4261, Z -4.6667, A 0.000, B 0.000, C 0.000 }
gfCNCPoint3[24699] = {X 270.7085, Y 11.2839, Z -4.6667, A 0.000, B 0.000, C 0.000 }
gfCNCPoint3[24700] = {X 270.8110, Y 12.1867, Z -4.6667, A 0.000, B 0.000, C 0.000 }
gfCNCPoint3[24701] = {X 270.8108, Y 13.0200, Z -4.6667, A 0.000, B 0.000, C 0.000 }
gfCNCPoint3[24702] = {X 270.7023, Y 13.9137, Z -4.6667, A 0.000, B 0.000, C 0.000 }
gfCNCPoint3[24703] = {X 270.4004, Y 14.7619, Z -4.6667, A 0.000, B 0.000, C 0.000 }
gfCNCPoint3[24704] = {X 269.9198, Y 15.5232, Z -4.6667, A 0.000, B 0.000, C 0.000 }
gfCNCPoint3[24705] = {X 269.2840, Y 16.1606, Z -4.6667, A 0.000, B 0.000, C 0.000 }
gfCNCPoint3[24706] = {X 269.2839, Y 28.5936, Z -4.6667, A 0.000, B 0.000, C 0.000 }
gfCNCPoint3[24707] = {X 273.2839, Y 28.5936, Z -4.6667, A 0.000, B 0.000, C 0.000 }
gfCNCPoint3[24708] = {X 269.2039, Y 28.5936, Z -4.6667, A 0.000, B 0.000, C 0.000 }
gfCNCPoint3[24709] = {X 269.2039, Y 41.0658, Z -4.6667, A 0.000, B 0.000, C 0.000 }
gfCNCPoint3[24710] = {X 269.3427, Y 41.1791, Z -4.6667, A 0.000, B 0.000, C 0.000 }
gfCNCPoint3[24711] = {X 269.9286, Y 41.8055, Z -4.6667, A 0.000, B 0.000, C 0.000 }
gfCNCPoint3[24712] = {X 270.3674, Y 42.5425, Z -4.6667, A 0.000, B 0.000, C 0.000 }
gfCNCPoint3[24713] = {X 270.6391, Y 43.3561, Z -4.6667, A 0.000, B 0.000, C 0.000 }
gfCNCPoint3[24714] = {X 270.7310, Y 44.2089, Z -4.6667, A 0.000, B 0.000, C 0.000 }
gfCNCPoint3[24715] = {X 270.7310, Y 45.0000, Z -4.6667, A 0.000, B 0.000, C 0.000 }
gfCNCPoint3[24716] = {X 270.6307, Y 45.8901, Z -4.6667, A 0.000, B 0.000, C 0.000 }
gfCNCPoint3[24717] = {X 270.3349, Y 46.7355, Z -4.6667, A 0.000, B 0.000, C 0.000 }
gfCNCPoint3[24718] = {X 269.8584, Y 47.4940, Z -4.6667, A 0.000, B 0.000, C 0.000 }
gfCNCPoint3[24719] = {X 269.2250, Y 48.1273, Z -4.6667, A 0.000, B 0.000, C 0.000 }
gfCNCPoint3[24720] = {X 268.4666, Y 48.6039, Z -4.6667, A 0.000, B 0.000, C 0.000 }
gfCNCPoint3[24721] = {X 267.6211, Y 48.8997, Z -4.6667, A 0.000, B 0.000, C 0.000 }
gfCNCPoint3[24722] = {X 266.7310, Y 49.0000, Z -4.6667, A 0.000, B 0.000, C 0.000 }
gfCNCPoint3[24723] = {X 260.2876, Y 49.0000, Z -4.6667, A 0.000, B 0.000, C 0.000 }
gfCNCPoint3[24724] = {X 259.3975, Y 48.8997, Z -4.6667, A 0.000, B 0.000, C 0.000 }
gfCNCPoint3[24725] = {X 258.5520, Y 48.6039, Z -4.6667, A 0.000, B 0.000, C 0.000 }
gfCNCPoint3[24726] = {X 257.7936, Y 48.1273, Z -4.6667, A 0.000, B 0.000, C 0.000 }
gfCNCPoint3[24727] = {X 257.1602, Y 47.4939, Z -4.6667, A 0.000, B 0.000, C 0.000 }
gfCNCPoint3[24728] = {X 256.6837, Y 46.7355, Z -4.6667, A 0.000, B 0.000, C 0.000 }
gfCNCPoint3[24729] = {X 256.3878, Y 45.8901, Z -4.6667, A 0.000, B 0.000, C 0.000 }
gfCNCPoint3[24730] = {X 256.2876, Y 45.0000, Z -4.6667, A 0.000, B 0.000, C 0.000 }
gfCNCPoint3[24731] = {X 256.2879, Y 44.1538, Z -4.6667, A 0.000, B 0.000, C 0.000 }
gfCNCPoint3[24732] = {X 256.3986, Y 43.2730, Z -4.6667, A 0.000, B 0.000, C 0.000 }
gfCNCPoint3[24733] = {X 256.7008, Y 42.4382, Z -4.6667, A 0.000, B 0.000, C 0.000 }
gfCNCPoint3[24734] = {X 257.1796, Y 41.6907, Z -4.6667, A 0.000, B 0.000, C 0.000 }
gfCNCPoint3[24735] = {X 257.8115, Y 41.0672, Z -4.6667, A 0.000, B 0.000, C 0.000 }
gfCNCPoint3[24736] = {X 257.8115, Y 34.1538, Z -4.6667, A 0.000, B 0.000, C 0.000 }
gfCNCPoint3[24737] = {X 254.8166, Y 34.1538, Z -4.6667, A 0.000, B 0.000, C 0.000 }
gfCNCPoint3[24738] = {X 254.5731, Y 34.1523, Z -4.6667, A 0.000, B 0.000, C 0.000 }
gfCNCPoint3[24739] = {X 250.1357, Y 42.7959, Z -4.6667, A 0.000, B 0.000, C 0.000 }
gfCNCPoint3[24740] = {X 250.3286, Y 43.4907, Z -4.6667, A 0.000, B 0.000, C 0.000 }
gfCNCPoint3[24741] = {X 250.3936, Y 44.2089, Z -4.6667, A 0.000, B 0.000, C 0.000 }
gfCNCPoint3[24742] = {X 250.3936, Y 45.0000, Z -4.6667, A 0.000, B 0.000, C 0.000 }
gfCNCPoint3[24743] = {X 250.2933, Y 45.8901, Z -4.6667, A 0.000, B 0.000, C 0.000 }
gfCNCPoint3[24744] = {X 249.9974, Y 46.7355, Z -4.6667, A 0.000, B 0.000, C 0.000 }
gfCNCPoint3[24745] = {X 249.5209, Y 47.4940, Z -4.6667, A 0.000, B 0.000, C 0.000 }
gfCNCPoint3[24746] = {X 248.8875, Y 48.1273, Z -4.6667, A 0.000, B 0.000, C 0.000 }
gfCNCPoint3[24747] = {X 248.1291, Y 48.6039, Z -4.6667, A 0.000, B 0.000, C 0.000 }
gfCNCPoint3[24748] = {X 247.2836, Y 48.8997, Z -4.6667, A 0.000, B 0.000, C 0.000 }
gfCNCPoint3[24749] = {X 246.3936, Y 49.0000, Z -4.6667, A 0.000, B 0.000, C 0.000 }
gfCNCPoint3[24750] = {X 239.8075, Y 49.0000, Z -4.6667, A 0.000, B 0.000, C 0.000 }
gfCNCPoint3[24751] = {X 238.9174, Y 48.8997, Z -4.6667, A 0.000, B 0.000, C 0.000 }
gfCNCPoint3[24752] = {X 238.0720, Y 48.6039, Z -4.6667, A 0.000, B 0.000, C 0.000 }
gfCNCPoint3[24753] = {X 237.3135, Y 48.1273, Z -4.6667, A 0.000, B 0.000, C 0.000 }
gfCNCPoint3[24754] = {X 236.6802, Y 47.4940, Z -4.6667, A 0.000, B 0.000, C 0.000 }
gfCNCPoint3[24755] = {X 236.2036, Y 46.7355, Z -4.6667, A 0.000, B 0.000, C 0.000 }
gfCNCPoint3[24756] = {X 235.9078, Y 45.8901, Z -4.6667, A 0.000, B 0.000, C 0.000 }
gfCNCPoint3[24757] = {X 235.8075, Y 45.0000, Z -4.6667, A 0.000, B 0.000, C 0.000 }
gfCNCPoint3[24758] = {X 235.8079, Y 44.1538, Z -4.6667, A 0.000, B 0.000, C 0.000 }
gfCNCPoint3[24759] = {X 235.9027, Y 43.3414, Z -4.6667, A 0.000, B 0.000, C 0.000 }
gfCNCPoint3[24760] = {X 236.1607, Y 42.5654, Z -4.6667, A 0.000, B 0.000, C 0.000 }
gfCNCPoint3[24761] = {X 236.5712, Y 41.8580, Z -4.6667, A 0.000, B 0.000, C 0.000 }
gfCNCPoint3[24762] = {X 237.1169, Y 41.2489, Z -4.6667, A 0.000, B 0.000, C 0.000 }
gfCNCPoint3[24763] = {X 237.7752, Y 40.7635, Z -4.6667, A 0.000, B 0.000, C 0.000 }
gfCNCPoint3[24764] = {X 238.5184, Y 40.4222, Z -4.6667, A 0.000, B 0.000, C 0.000 }
gfCNCPoint3[24765] = {X 242.7046, Y 32.2282, Z -4.6667, A 0.000, B 0.000, C 0.000 }
gfCNCPoint3[24766] = {X 241.5064, Y 31.4659, Z -4.6667, A 0.000, B 0.000, C 0.000 }
gfCNCPoint3[24767] = {X 240.4164, Y 30.5556, Z -4.6667, A 0.000, B 0.000, C 0.000 }
gfCNCPoint3[24768] = {X 239.4528, Y 29.5124, Z -4.6667, A 0.000, B 0.000, C 0.000 }
gfCNCPoint3[24769] = {X 238.6317, Y 28.3537, Z -4.6667, A 0.000, B 0.000, C 0.000 }
gfCNCPoint3[24770] = {X 237.9667, Y 27.0989, Z -4.6667, A 0.000, B 0.000, C 0.000 }
gfCNCPoint3[24771] = {X 237.4689, Y 25.7689, Z -4.6667, A 0.000, B 0.000, C 0.000 }
gfCNCPoint3[24772] = {X 237.0573, Y 23.9929, Z -4.6667, A 0.000, B 0.000, C 0.000 }
gfCNCPoint3[24773] = {X 236.8476, Y 22.1820, Z -4.6667, A 0.000, B 0.000, C 0.000 }
gfCNCPoint3[24774] = {X 236.8426, Y 20.3590, Z -4.6667, A 0.000, B 0.000, C 0.000 }
gfCNCPoint3[24775] = {X 237.0422, Y 18.5469, Z -4.6667, A 0.000, B 0.000, C 0.000 }
gfCNCPoint3[24776] = {X 237.4439, Y 16.7687, Z -4.6667, A 0.000, B 0.000, C 0.000 }
gfCNCPoint3[24777] = {X 237.9989, Y 15.2353, Z -4.6667, A 0.000, B 0.000, C 0.000 }
gfCNCPoint3[24778] = {X 238.7648, Y 13.7956, Z -4.6667, A 0.000, B 0.000, C 0.000 }
gfCNCPoint3[24779] = {X 239.7262, Y 12.4783, Z -4.6667, A 0.000, B 0.000, C 0.000 }
gfCNCPoint3[24780] = {X 240.8638, Y 11.3098, Z -4.6667, A 0.000, B 0.000, C 0.000 }
gfCNCPoint3[24781] = {X 242.1550, Y 10.3136, Z -4.6667, A 0.000, B 0.000, C 0.000 }
gfCNCPoint3[24782] = {X 243.5737, Y 9.5095, Z -4.6667, A 0.000, B 0.000, C 0.000 }
gfCNCPoint3[24783] = {X 245.0918, Y 8.9137, Z -4.6667, A 0.000, B 0.000, C 0.000 }
gfCNCPoint3[24784] = {X 246.6787, Y 8.5381, Z -4.6667, A 0.000, B 0.000, C 0.000 }
gfCNCPoint3[24785] = {X 248.7483, Y 8.2700, Z -4.6667, A 0.000, B 0.000, C 0.000 }
gfCNCPoint3[24786] = {X 250.8336, Y 8.1906, Z -4.6667, A 0.000, B 0.000, C 0.000 }
gfCNCPoint3[24787] = {X 266.7608, Y 8.1906, Z -4.6667, A 0.000, B 0.000, C 0.000 }
gfCNCPoint3[24788] = {X 267.6452, Y 8.2968, Z -4.6667, A 0.000, B 0.000, C 0.000 }
gfCNCPoint3[24789] = {X 268.4843, Y 8.5961, Z -4.6667, A 0.000, B 0.000, C 0.000 }
gfCNCPoint3[24790] = {X 269.2364, Y 9.0736, Z -4.6667, A 0.000, B 0.000, C 0.000 }
gfCNCPoint3[24791] = {X 269.8642, Y 9.7055, Z -4.6667, A 0.000, B 0.000, C 0.000 }
gfCNCPoint3[24792] = {X 270.3368, Y 10.4607, Z -4.6667, A 0.000, B 0.000, C 0.000 }
gfCNCPoint3[24793] = {X 270.6305, Y 11.3017, Z -4.6667, A 0.000, B 0.000, C 0.000 }
gfCNCPoint3[24794] = {X 270.7310, Y 12.1869, Z -4.6667, A 0.000, B 0.000, C 0.000 }
gfCNCPoint3[24795] = {X 270.7308, Y 13.0192, Z -4.6667, A 0.000, B 0.000, C 0.000 }
gfCNCPoint3[24796] = {X 270.6222, Y 13.9047, Z -4.6667, A 0.000, B 0.000, C 0.000 }
gfCNCPoint3[24797] = {X 270.3200, Y 14.7441, Z -4.6667, A 0.000, B 0.000, C 0.000 }
gfCNCPoint3[24798] = {X 269.8394, Y 15.4956, Z -4.6667, A 0.000, B 0.000, C 0.000 }
gfCNCPoint3[24799] = {X 269.2040, Y 16.1219, Z -4.6667, A 0.000, B 0.000, C 0.000 }
gfCNCPoint3[24800] = {X 269.2039, Y 28.5936, Z -4.6667, A 0.000, B 0.000, C 0.000 }
gfCNCPoint3[24801] = {X 273.2839, Y 28.5936, Z -4.6667, A 0.000, B 0.000, C 0.000 }
gfCNCPoint3[24802] = {X 273.2839, Y 28.5936, Z -1.6667, A 0.000, B 0.000, C 0.000 }
gfCNCPoint3[24803] = {X 273.2839, Y 28.5936, Z 11.0000, A 0.000, B 0.000, C 0.000 }
gfCNCPoint3[24804] = {X 277.7451, Y 28.5925, Z 11.0000, A 0.000, B 0.000, C 0.000 }
gfCNCPoint3[24805] = {X 277.7451, Y 28.5925, Z -1.6667, A 0.000, B 0.000, C 0.000 }
gfCNCPoint3[24806] = {X 277.7451, Y 28.5925, Z -4.6667, A 0.000, B 0.000, C 0.000 }
gfCNCPoint3[24807] = {X 281.8251, Y 28.5924, Z -4.6667, A 0.000, B 0.000, C 0.000 }
gfCNCPoint3[24808] = {X 281.8249, Y 16.2739, Z -4.6667, A 0.000, B 0.000, C 0.000 }
gfCNCPoint3[24809] = {X 281.1865, Y 15.6028, Z -4.6667, A 0.000, B 0.000, C 0.000 }
gfCNCPoint3[24810] = {X 280.7059, Y 14.8111, Z -4.6667, A 0.000, B 0.000, C 0.000 }
gfCNCPoint3[24811] = {X 280.4050, Y 13.9351, Z -4.6667, A 0.000, B 0.000, C 0.000 }
gfCNCPoint3[24812] = {X 280.2978, Y 13.0151, Z -4.6667, A 0.000, B 0.000, C 0.000 }
gfCNCPoint3[24813] = {X 280.2977, Y 12.1868, Z -4.6667, A 0.000, B 0.000, C 0.000 }
gfCNCPoint3[24814] = {X 280.4060, Y 11.2255, Z -4.6667, A 0.000, B 0.000, C 0.000 }
gfCNCPoint3[24815] = {X 280.7255, Y 10.3124, Z -4.6667, A 0.000, B 0.000, C 0.000 }
gfCNCPoint3[24816] = {X 281.2402, Y 9.4933, Z -4.6667, A 0.000, B 0.000, C 0.000 }
gfCNCPoint3[24817] = {X 281.9242, Y 8.8093, Z -4.6667, A 0.000, B 0.000, C 0.000 }
gfCNCPoint3[24818] = {X 282.7433, Y 8.2946, Z -4.6667, A 0.000, B 0.000, C 0.000 }
gfCNCPoint3[24819] = {X 283.6564, Y 7.9751, Z -4.6667, A 0.000, B 0.000, C 0.000 }
gfCNCPoint3[24820] = {X 284.6177, Y 7.8668, Z -4.6667, A 0.000, B 0.000, C 0.000 }
gfCNCPoint3[24821] = {X 291.0611, Y 7.8668, Z -4.6667, A 0.000, B 0.000, C 0.000 }
gfCNCPoint3[24822] = {X 292.0224, Y 7.9751, Z -4.6667, A 0.000, B 0.000, C 0.000 }
gfCNCPoint3[24823] = {X 292.9355, Y 8.2946, Z -4.6667, A 0.000, B 0.000, C 0.000 }
gfCNCPoint3[24824] = {X 293.7546, Y 8.8093, Z -4.6667, A 0.000, B 0.000, C 0.000 }
gfCNCPoint3[24825] = {X 294.4386, Y 9.4933, Z -4.6667, A 0.000, B 0.000, C 0.000 }
gfCNCPoint3[24826] = {X 294.9533, Y 10.3124, Z -4.6667, A 0.000, B 0.000, C 0.000 }
gfCNCPoint3[24827] = {X 295.2728, Y 11.2255, Z -4.6667, A 0.000, B 0.000, C 0.000 }
gfCNCPoint3[24828] = {X 295.3811, Y 12.1868, Z -4.6667, A 0.000, B 0.000, C 0.000 }
gfCNCPoint3[24829] = {X 295.3811, Y 12.9782, Z -4.6667, A 0.000, B 0.000, C 0.000 }
gfCNCPoint3[24830] = {X 295.2797, Y 13.9081, Z -4.6667, A 0.000, B 0.000, C 0.000 }
gfCNCPoint3[24831] = {X 294.9806, Y 14.7943, Z -4.6667, A 0.000, B 0.000, C 0.000 }
gfCNCPoint3[24832] = {X 294.4976, Y 15.5954, Z -4.6667, A 0.000, B 0.000, C 0.000 }
gfCNCPoint3[24833] = {X 293.8536, Y 16.2738, Z -4.6667, A 0.000, B 0.000, C 0.000 }
gfCNCPoint3[24834] = {X 293.8547, Y 22.1965, Z -4.6667, A 0.000, B 0.000, C 0.000 }
gfCNCPoint3[24835] = {X 302.7591, Y 22.1965, Z -4.6667, A 0.000, B 0.000, C 0.000 }
gfCNCPoint3[24836] = {X 302.7641, Y 16.2778, Z -4.6667, A 0.000, B 0.000, C 0.000 }
gfCNCPoint3[24837] = {X 302.1241, Y 15.6067, Z -4.6667, A 0.000, B 0.000, C 0.000 }
gfCNCPoint3[24838] = {X 301.6420, Y 14.8145, Z -4.6667, A 0.000, B 0.000, C 0.000 }
gfCNCPoint3[24839] = {X 301.3402, Y 13.9376, Z -4.6667, A 0.000, B 0.000, C 0.000 }
gfCNCPoint3[24840] = {X 301.2324, Y 13.0165, Z -4.6667, A 0.000, B 0.000, C 0.000 }
gfCNCPoint3[24841] = {X 301.2323, Y 12.1868, Z -4.6667, A 0.000, B 0.000, C 0.000 }
gfCNCPoint3[24842] = {X 301.3406, Y 11.2255, Z -4.6667, A 0.000, B 0.000, C 0.000 }
gfCNCPoint3[24843] = {X 301.6601, Y 10.3124, Z -4.6667, A 0.000, B 0.000, C 0.000 }
gfCNCPoint3[24844] = {X 302.1747, Y 9.4933, Z -4.6667, A 0.000, B 0.000, C 0.000 }
gfCNCPoint3[24845] = {X 302.8588, Y 8.8093, Z -4.6667, A 0.000, B 0.000, C 0.000 }
gfCNCPoint3[24846] = {X 303.6779, Y 8.2946, Z -4.6667, A 0.000, B 0.000, C 0.000 }
gfCNCPoint3[24847] = {X 304.5910, Y 7.9751, Z -4.6667, A 0.000, B 0.000, C 0.000 }
gfCNCPoint3[24848] = {X 305.5523, Y 7.8668, Z -4.6667, A 0.000, B 0.000, C 0.000 }
gfCNCPoint3[24849] = {X 311.9957, Y 7.8668, Z -4.6667, A 0.000, B 0.000, C 0.000 }
gfCNCPoint3[24850] = {X 312.9570, Y 7.9751, Z -4.6667, A 0.000, B 0.000, C 0.000 }
gfCNCPoint3[24851] = {X 313.8701, Y 8.2946, Z -4.6667, A 0.000, B 0.000, C 0.000 }
gfCNCPoint3[24852] = {X 314.6892, Y 8.8093, Z -4.6667, A 0.000, B 0.000, C 0.000 }
gfCNCPoint3[24853] = {X 315.3732, Y 9.4933, Z -4.6667, A 0.000, B 0.000, C 0.000 }
gfCNCPoint3[24854] = {X 315.8879, Y 10.3124, Z -4.6667, A 0.000, B 0.000, C 0.000 }
gfCNCPoint3[24855] = {X 316.2074, Y 11.2255, Z -4.6667, A 0.000, B 0.000, C 0.000 }
gfCNCPoint3[24856] = {X 316.3157, Y 12.1868, Z -4.6667, A 0.000, B 0.000, C 0.000 }
gfCNCPoint3[24857] = {X 316.3157, Y 12.9782, Z -4.6667, A 0.000, B 0.000, C 0.000 }
gfCNCPoint3[24858] = {X 316.2145, Y 13.9077, Z -4.6667, A 0.000, B 0.000, C 0.000 }
gfCNCPoint3[24859] = {X 315.9156, Y 14.7937, Z -4.6667, A 0.000, B 0.000, C 0.000 }
gfCNCPoint3[24860] = {X 315.4331, Y 15.5947, Z -4.6667, A 0.000, B 0.000, C 0.000 }
gfCNCPoint3[24861] = {X 314.7895, Y 16.2730, Z -4.6667, A 0.000, B 0.000, C 0.000 }
gfCNCPoint3[24862] = {X 314.7881, Y 40.9126, Z -4.6667, A 0.000, B 0.000, C 0.000 }
gfCNCPoint3[24863] = {X 315.4266, Y 41.5836, Z -4.6667, A 0.000, B 0.000, C 0.000 }
gfCNCPoint3[24864] = {X 315.9073, Y 42.3753, Z -4.6667, A 0.000, B 0.000, C 0.000 }
gfCNCPoint3[24865] = {X 316.2083, Y 43.2513, Z -4.6667, A 0.000, B 0.000, C 0.000 }
gfCNCPoint3[24866] = {X 316.3156, Y 44.1713, Z -4.6667, A 0.000, B 0.000, C 0.000 }
gfCNCPoint3[24867] = {X 316.3157, Y 45.0000, Z -4.6667, A 0.000, B 0.000, C 0.000 }
gfCNCPoint3[24868] = {X 316.2074, Y 45.9613, Z -4.6667, A 0.000, B 0.000, C 0.000 }
gfCNCPoint3[24869] = {X 315.8879, Y 46.8744, Z -4.6667, A 0.000, B 0.000, C 0.000 }
gfCNCPoint3[24870] = {X 315.3732, Y 47.6935, Z -4.6667, A 0.000, B 0.000, C 0.000 }
gfCNCPoint3[24871] = {X 314.6892, Y 48.3775, Z -4.6667, A 0.000, B 0.000, C 0.000 }
gfCNCPoint3[24872] = {X 313.8701, Y 48.8922, Z -4.6667, A 0.000, B 0.000, C 0.000 }
gfCNCPoint3[24873] = {X 312.9570, Y 49.2117, Z -4.6667, A 0.000, B 0.000, C 0.000 }
gfCNCPoint3[24874] = {X 311.9957, Y 49.3200, Z -4.6667, A 0.000, B 0.000, C 0.000 }
gfCNCPoint3[24875] = {X 305.5523, Y 49.3200, Z -4.6667, A 0.000, B 0.000, C 0.000 }
gfCNCPoint3[24876] = {X 304.5958, Y 49.2128, Z -4.6667, A 0.000, B 0.000, C 0.000 }
gfCNCPoint3[24877] = {X 303.6868, Y 48.8965, Z -4.6667, A 0.000, B 0.000, C 0.000 }
gfCNCPoint3[24878] = {X 302.8704, Y 48.3868, Z -4.6667, A 0.000, B 0.000, C 0.000 }
gfCNCPoint3[24879] = {X 302.1872, Y 47.7090, Z -4.6667, A 0.000, B 0.000, C 0.000 }
gfCNCPoint3[24880] = {X 301.6709, Y 46.8967, Z -4.6667, A 0.000, B 0.000, C 0.000 }
gfCNCPoint3[24881] = {X 301.3473, Y 45.9903, Z -4.6667, A 0.000, B 0.000, C 0.000 }
gfCNCPoint3[24882] = {X 301.2324, Y 45.0348, Z -4.6667, A 0.000, B 0.000, C 0.000 }
gfCNCPoint3[24883] = {X 301.2323, Y 44.2012, Z -4.6667, A 0.000, B 0.000, C 0.000 }
gfCNCPoint3[24884] = {X 301.3499, Y 43.2652, Z -4.6667, A 0.000, B 0.000, C 0.000 }
gfCNCPoint3[24885] = {X 301.6531, Y 42.3718, Z -4.6667, A 0.000, B 0.000, C 0.000 }
gfCNCPoint3[24886] = {X 302.1295, Y 41.5574, Z -4.6667, A 0.000, B 0.000, C 0.000 }
gfCNCPoint3[24887] = {X 302.7597, Y 40.8554, Z -4.6667, A 0.000, B 0.000, C 0.000 }
gfCNCPoint3[24888] = {X 302.7597, Y 34.0343, Z -4.6667, A 0.000, B 0.000, C 0.000 }
gfCNCPoint3[24889] = {X 293.8545, Y 34.0343, Z -4.6667, A 0.000, B 0.000, C 0.000 }
gfCNCPoint3[24890] = {X 293.8537, Y 40.9023, Z -4.6667, A 0.000, B 0.000, C 0.000 }
gfCNCPoint3[24891] = {X 294.4928, Y 41.5863, Z -4.6667, A 0.000, B 0.000, C 0.000 }
gfCNCPoint3[24892] = {X 294.9734, Y 42.3896, Z -4.6667, A 0.000, B 0.000, C 0.000 }
gfCNCPoint3[24893] = {X 295.2740, Y 43.2762, Z -4.6667, A 0.000, B 0.000, C 0.000 }
gfCNCPoint3[24894] = {X 295.3811, Y 44.2062, Z -4.6667, A 0.000, B 0.000, C 0.000 }
gfCNCPoint3[24895] = {X 295.3811, Y 45.0000, Z -4.6667, A 0.000, B 0.000, C 0.000 }
gfCNCPoint3[24896] = {X 295.2728, Y 45.9613, Z -4.6667, A 0.000, B 0.000, C 0.000 }
gfCNCPoint3[24897] = {X 294.9533, Y 46.8744, Z -4.6667, A 0.000, B 0.000, C 0.000 }
gfCNCPoint3[24898] = {X 294.4386, Y 47.6935, Z -4.6667, A 0.000, B 0.000, C 0.000 }
gfCNCPoint3[24899] = {X 293.7546, Y 48.3775, Z -4.6667, A 0.000, B 0.000, C 0.000 }
gfCNCPoint3[24900] = {X 292.9355, Y 48.8922, Z -4.6667, A 0.000, B 0.000, C 0.000 }
gfCNCPoint3[24901] = {X 292.0224, Y 49.2117, Z -4.6667, A 0.000, B 0.000, C 0.000 }
gfCNCPoint3[24902] = {X 291.0611, Y 49.3200, Z -4.6667, A 0.000, B 0.000, C 0.000 }
gfCNCPoint3[24903] = {X 284.6177, Y 49.3200, Z -4.6667, A 0.000, B 0.000, C 0.000 }
gfCNCPoint3[24904] = {X 283.6613, Y 49.2128, Z -4.6667, A 0.000, B 0.000, C 0.000 }
gfCNCPoint3[24905] = {X 282.7524, Y 48.8965, Z -4.6667, A 0.000, B 0.000, C 0.000 }
gfCNCPoint3[24906] = {X 281.9360, Y 48.3869, Z -4.6667, A 0.000, B 0.000, C 0.000 }
gfCNCPoint3[24907] = {X 281.2527, Y 47.7092, Z -4.6667, A 0.000, B 0.000, C 0.000 }
gfCNCPoint3[24908] = {X 280.7365, Y 46.8970, Z -4.6667, A 0.000, B 0.000, C 0.000 }
gfCNCPoint3[24909] = {X 280.4128, Y 45.9907, Z -4.6667, A 0.000, B 0.000, C 0.000 }
gfCNCPoint3[24910] = {X 280.2978, Y 45.0352, Z -4.6667, A 0.000, B 0.000, C 0.000 }
gfCNCPoint3[24911] = {X 280.2977, Y 44.2072, Z -4.6667, A 0.000, B 0.000, C 0.000 }
gfCNCPoint3[24912] = {X 280.4025, Y 43.2782, Z -4.6667, A 0.000, B 0.000, C 0.000 }
gfCNCPoint3[24913] = {X 280.7026, Y 42.3927, Z -4.6667, A 0.000, B 0.000, C 0.000 }
gfCNCPoint3[24914] = {X 281.1842, Y 41.5914, Z -4.6667, A 0.000, B 0.000, C 0.000 }
gfCNCPoint3[24915] = {X 281.8253, Y 40.9109, Z -4.6667, A 0.000, B 0.000, C 0.000 }
gfCNCPoint3[24916] = {X 281.8251, Y 28.5924, Z -4.6667, A 0.000, B 0.000, C 0.000 }
gfCNCPoint3[24917] = {X 277.8251, Y 28.5925, Z -4.6667, A 0.000, B 0.000, C 0.000 }
gfCNCPoint3[24918] = {X 281.9051, Y 28.5924, Z -4.6667, A 0.000, B 0.000, C 0.000 }
gfCNCPoint3[24919] = {X 281.9049, Y 16.2366, Z -4.6667, A 0.000, B 0.000, C 0.000 }
gfCNCPoint3[24920] = {X 281.2670, Y 15.5762, Z -4.6667, A 0.000, B 0.000, C 0.000 }
gfCNCPoint3[24921] = {X 280.7862, Y 14.7938, Z -4.6667, A 0.000, B 0.000, C 0.000 }
gfCNCPoint3[24922] = {X 280.4851, Y 13.9264, Z -4.6667, A 0.000, B 0.000, C 0.000 }
gfCNCPoint3[24923] = {X 280.3778, Y 13.0144, Z -4.6667, A 0.000, B 0.000, C 0.000 }
gfCNCPoint3[24924] = {X 280.3777, Y 12.1868, Z -4.6667, A 0.000, B 0.000, C 0.000 }
gfCNCPoint3[24925] = {X 280.4840, Y 11.2433, Z -4.6667, A 0.000, B 0.000, C 0.000 }
gfCNCPoint3[24926] = {X 280.7976, Y 10.3472, Z -4.6667, A 0.000, B 0.000, C 0.000 }
gfCNCPoint3[24927] = {X 281.3027, Y 9.5432, Z -4.6667, A 0.000, B 0.000, C 0.000 }
gfCNCPoint3[24928] = {X 281.9741, Y 8.8719, Z -4.6667, A 0.000, B 0.000, C 0.000 }
gfCNCPoint3[24929] = {X 282.7780, Y 8.3667, Z -4.6667, A 0.000, B 0.000, C 0.000 }
gfCNCPoint3[24930] = {X 283.6742, Y 8.0531, Z -4.6667, A 0.000, B 0.000, C 0.000 }
gfCNCPoint3[24931] = {X 284.6177, Y 7.9468, Z -4.6667, A 0.000, B 0.000, C 0.000 }
gfCNCPoint3[24932] = {X 291.0611, Y 7.9468, Z -4.6667, A 0.000, B 0.000, C 0.000 }
gfCNCPoint3[24933] = {X 292.0046, Y 8.0531, Z -4.6667, A 0.000, B 0.000, C 0.000 }
gfCNCPoint3[24934] = {X 292.9008, Y 8.3667, Z -4.6667, A 0.000, B 0.000, C 0.000 }
gfCNCPoint3[24935] = {X 293.7047, Y 8.8718, Z -4.6667, A 0.000, B 0.000, C 0.000 }
gfCNCPoint3[24936] = {X 294.3761, Y 9.5432, Z -4.6667, A 0.000, B 0.000, C 0.000 }
gfCNCPoint3[24937] = {X 294.8812, Y 10.3471, Z -4.6667, A 0.000, B 0.000, C 0.000 }
gfCNCPoint3[24938] = {X 295.1948, Y 11.2433, Z -4.6667, A 0.000, B 0.000, C 0.000 }
gfCNCPoint3[24939] = {X 295.3011, Y 12.1868, Z -4.6667, A 0.000, B 0.000, C 0.000 }
gfCNCPoint3[24940] = {X 295.3011, Y 12.9782, Z -4.6667, A 0.000, B 0.000, C 0.000 }
gfCNCPoint3[24941] = {X 295.1996, Y 13.8998, Z -4.6667, A 0.000, B 0.000, C 0.000 }
gfCNCPoint3[24942] = {X 294.9002, Y 14.7774, Z -4.6667, A 0.000, B 0.000, C 0.000 }
gfCNCPoint3[24943] = {X 294.4171, Y 15.5689, Z -4.6667, A 0.000, B 0.000, C 0.000 }
gfCNCPoint3[24944] = {X 293.7736, Y 16.2365, Z -4.6667, A 0.000, B 0.000, C 0.000 }
gfCNCPoint3[24945] = {X 293.7747, Y 22.2765, Z -4.6667, A 0.000, B 0.000, C 0.000 }
gfCNCPoint3[24946] = {X 302.8391, Y 22.2765, Z -4.6667, A 0.000, B 0.000, C 0.000 }
gfCNCPoint3[24947] = {X 302.8441, Y 16.2405, Z -4.6667, A 0.000, B 0.000, C 0.000 }
gfCNCPoint3[24948] = {X 302.2045, Y 15.5800, Z -4.6667, A 0.000, B 0.000, C 0.000 }
gfCNCPoint3[24949] = {X 301.7223, Y 14.7972, Z -4.6667, A 0.000, B 0.000, C 0.000 }
gfCNCPoint3[24950] = {X 301.4202, Y 13.9289, Z -4.6667, A 0.000, B 0.000, C 0.000 }
gfCNCPoint3[24951] = {X 301.3124, Y 13.0158, Z -4.6667, A 0.000, B 0.000, C 0.000 }
gfCNCPoint3[24952] = {X 301.3123, Y 12.1868, Z -4.6667, A 0.000, B 0.000, C 0.000 }
gfCNCPoint3[24953] = {X 301.4186, Y 11.2433, Z -4.6667, A 0.000, B 0.000, C 0.000 }
gfCNCPoint3[24954] = {X 301.7321, Y 10.3471, Z -4.6667, A 0.000, B 0.000, C 0.000 }
gfCNCPoint3[24955] = {X 302.2373, Y 9.5432, Z -4.6667, A 0.000, B 0.000, C 0.000 }
gfCNCPoint3[24956] = {X 302.9087, Y 8.8718, Z -4.6667, A 0.000, B 0.000, C 0.000 }
gfCNCPoint3[24957] = {X 303.7126, Y 8.3667, Z -4.6667, A 0.000, B 0.000, C 0.000 }
gfCNCPoint3[24958] = {X 304.6088, Y 8.0531, Z -4.6667, A 0.000, B 0.000, C 0.000 }
gfCNCPoint3[24959] = {X 305.5523, Y 7.9468, Z -4.6667, A 0.000, B 0.000, C 0.000 }
gfCNCPoint3[24960] = {X 311.9957, Y 7.9468, Z -4.6667, A 0.000, B 0.000, C 0.000 }
gfCNCPoint3[24961] = {X 312.9392, Y 8.0531, Z -4.6667, A 0.000, B 0.000, C 0.000 }
gfCNCPoint3[24962] = {X 313.8354, Y 8.3667, Z -4.6667, A 0.000, B 0.000, C 0.000 }
gfCNCPoint3[24963] = {X 314.6393, Y 8.8718, Z -4.6667, A 0.000, B 0.000, C 0.000 }
gfCNCPoint3[24964] = {X 315.3107, Y 9.5432, Z -4.6667, A 0.000, B 0.000, C 0.000 }
gfCNCPoint3[24965] = {X 315.8158, Y 10.3471, Z -4.6667, A 0.000, B 0.000, C 0.000 }
gfCNCPoint3[24966] = {X 316.1294, Y 11.2433, Z -4.6667, A 0.000, B 0.000, C 0.000 }
gfCNCPoint3[24967] = {X 316.2357, Y 12.1868, Z -4.6667, A 0.000, B 0.000, C 0.000 }
gfCNCPoint3[24968] = {X 316.2357, Y 12.9782, Z -4.6667, A 0.000, B 0.000, C 0.000 }
gfCNCPoint3[24969] = {X 316.1344, Y 13.8995, Z -4.6667, A 0.000, B 0.000, C 0.000 }
gfCNCPoint3[24970] = {X 315.8352, Y 14.7768, Z -4.6667, A 0.000, B 0.000, C 0.000 }
gfCNCPoint3[24971] = {X 315.3526, Y 15.5682, Z -4.6667, A 0.000, B 0.000, C 0.000 }
gfCNCPoint3[24972] = {X 314.7095, Y 16.2358, Z -4.6667, A 0.000, B 0.000, C 0.000 }
gfCNCPoint3[24973] = {X 314.7081, Y 40.9509, Z -4.6667, A 0.000, B 0.000, C 0.000 }
gfCNCPoint3[24974] = {X 314.7364, Y 40.9736, Z -4.6667, A 0.000, B 0.000, C 0.000 }
gfCNCPoint3[24975] = {X 315.3630, Y 41.6322, Z -4.6667, A 0.000, B 0.000, C 0.000 }
gfCNCPoint3[24976] = {X 315.8349, Y 42.4092, Z -4.6667, A 0.000, B 0.000, C 0.000 }
gfCNCPoint3[24977] = {X 316.1303, Y 43.2690, Z -4.6667, A 0.000, B 0.000, C 0.000 }
gfCNCPoint3[24978] = {X 316.2356, Y 44.1720, Z -4.6667, A 0.000, B 0.000, C 0.000 }
gfCNCPoint3[24979] = {X 316.2357, Y 45.0000, Z -4.6667, A 0.000, B 0.000, C 0.000 }
gfCNCPoint3[24980] = {X 316.1294, Y 45.9435, Z -4.6667, A 0.000, B 0.000, C 0.000 }
gfCNCPoint3[24981] = {X 315.8158, Y 46.8397, Z -4.6667, A 0.000, B 0.000, C 0.000 }
gfCNCPoint3[24982] = {X 315.3107, Y 47.6436, Z -4.6667, A 0.000, B 0.000, C 0.000 }
gfCNCPoint3[24983] = {X 314.6393, Y 48.3150, Z -4.6667, A 0.000, B 0.000, C 0.000 }
gfCNCPoint3[24984] = {X 313.8354, Y 48.8201, Z -4.6667, A 0.000, B 0.000, C 0.000 }
gfCNCPoint3[24985] = {X 312.9392, Y 49.1337, Z -4.6667, A 0.000, B 0.000, C 0.000 }
gfCNCPoint3[24986] = {X 311.9957, Y 49.2400, Z -4.6667, A 0.000, B 0.000, C 0.000 }
gfCNCPoint3[24987] = {X 305.5523, Y 49.2400, Z -4.6667, A 0.000, B 0.000, C 0.000 }
gfCNCPoint3[24988] = {X 304.6135, Y 49.1348, Z -4.6667, A 0.000, B 0.000, C 0.000 }
gfCNCPoint3[24989] = {X 303.7214, Y 48.8243, Z -4.6667, A 0.000, B 0.000, C 0.000 }
gfCNCPoint3[24990] = {X 302.9201, Y 48.3241, Z -4.6667, A 0.000, B 0.000, C 0.000 }
gfCNCPoint3[24991] = {X 302.2495, Y 47.6588, Z -4.6667, A 0.000, B 0.000, C 0.000 }
gfCNCPoint3[24992] = {X 301.7428, Y 46.8616, Z -4.6667, A 0.000, B 0.000, C 0.000 }
gfCNCPoint3[24993] = {X 301.4252, Y 45.9720, Z -4.6667, A 0.000, B 0.000, C 0.000 }
gfCNCPoint3[24994] = {X 301.3124, Y 45.0341, Z -4.6667, A 0.000, B 0.000, C 0.000 }
gfCNCPoint3[24995] = {X 301.3123, Y 44.2031, Z -4.6667, A 0.000, B 0.000, C 0.000 }
gfCNCPoint3[24996] = {X 301.4299, Y 43.2745, Z -4.6667, A 0.000, B 0.000, C 0.000 }
gfCNCPoint3[24997] = {X 301.7332, Y 42.3890, Z -4.6667, A 0.000, B 0.000, C 0.000 }
gfCNCPoint3[24998] = {X 302.2098, Y 41.5833, Z -4.6667, A 0.000, B 0.000, C 0.000 }
gfCNCPoint3[24999] = {X 302.8397, Y 40.8909, Z -4.6667, A 0.000, B 0.000, C 0.000 }
gfCNCPoint3[25000] = {X 302.8397, Y 33.9543, Z -4.6667, A 0.000, B 0.000, C 0.000 }
gfCNCPoint3[25001] = {X 293.7745, Y 33.9543, Z -4.6667, A 0.000, B 0.000, C 0.000 }
gfCNCPoint3[25002] = {X 293.7737, Y 40.9391, Z -4.6667, A 0.000, B 0.000, C 0.000 }
gfCNCPoint3[25003] = {X 294.4124, Y 41.6127, Z -4.6667, A 0.000, B 0.000, C 0.000 }
gfCNCPoint3[25004] = {X 294.8931, Y 42.4067, Z -4.6667, A 0.000, B 0.000, C 0.000 }
gfCNCPoint3[25005] = {X 295.1940, Y 43.2848, Z -4.6667, A 0.000, B 0.000, C 0.000 }
gfCNCPoint3[25006] = {X 295.3011, Y 44.2068, Z -4.6667, A 0.000, B 0.000, C 0.000 }
gfCNCPoint3[25007] = {X 295.3011, Y 45.0000, Z -4.6667, A 0.000, B 0.000, C 0.000 }
gfCNCPoint3[25008] = {X 295.1948, Y 45.9435, Z -4.6667, A 0.000, B 0.000, C 0.000 }
gfCNCPoint3[25009] = {X 294.8812, Y 46.8397, Z -4.6667, A 0.000, B 0.000, C 0.000 }
gfCNCPoint3[25010] = {X 294.3761, Y 47.6436, Z -4.6667, A 0.000, B 0.000, C 0.000 }
gfCNCPoint3[25011] = {X 293.7047, Y 48.3150, Z -4.6667, A 0.000, B 0.000, C 0.000 }
gfCNCPoint3[25012] = {X 292.9008, Y 48.8201, Z -4.6667, A 0.000, B 0.000, C 0.000 }
gfCNCPoint3[25013] = {X 292.0046, Y 49.1337, Z -4.6667, A 0.000, B 0.000, C 0.000 }
gfCNCPoint3[25014] = {X 291.0611, Y 49.2400, Z -4.6667, A 0.000, B 0.000, C 0.000 }
gfCNCPoint3[25015] = {X 284.6177, Y 49.2400, Z -4.6667, A 0.000, B 0.000, C 0.000 }
gfCNCPoint3[25016] = {X 283.6790, Y 49.1348, Z -4.6667, A 0.000, B 0.000, C 0.000 }
gfCNCPoint3[25017] = {X 282.7869, Y 48.8244, Z -4.6667, A 0.000, B 0.000, C 0.000 }
gfCNCPoint3[25018] = {X 281.9857, Y 48.3242, Z -4.6667, A 0.000, B 0.000, C 0.000 }
gfCNCPoint3[25019] = {X 281.3150, Y 47.6590, Z -4.6667, A 0.000, B 0.000, C 0.000 }
gfCNCPoint3[25020] = {X 280.8083, Y 46.8619, Z -4.6667, A 0.000, B 0.000, C 0.000 }
gfCNCPoint3[25021] = {X 280.4907, Y 45.9723, Z -4.6667, A 0.000, B 0.000, C 0.000 }
gfCNCPoint3[25022] = {X 280.3778, Y 45.0345, Z -4.6667, A 0.000, B 0.000, C 0.000 }
gfCNCPoint3[25023] = {X 280.3777, Y 44.2076, Z -4.6667, A 0.000, B 0.000, C 0.000 }
gfCNCPoint3[25024] = {X 280.4826, Y 43.2867, Z -4.6667, A 0.000, B 0.000, C 0.000 }
gfCNCPoint3[25025] = {X 280.7829, Y 42.4097, Z -4.6667, A 0.000, B 0.000, C 0.000 }
gfCNCPoint3[25026] = {X 281.2647, Y 41.6178, Z -4.6667, A 0.000, B 0.000, C 0.000 }
gfCNCPoint3[25027] = {X 281.9053, Y 40.9479, Z -4.6667, A 0.000, B 0.000, C 0.000 }
gfCNCPoint3[25028] = {X 281.9051, Y 28.5924, Z -4.6667, A 0.000, B 0.000, C 0.000 }
gfCNCPoint3[25029] = {X 277.9051, Y 28.5925, Z -4.6667, A 0.000, B 0.000, C 0.000 }
gfCNCPoint3[25030] = {X 281.9851, Y 28.5924, Z -4.6667, A 0.000, B 0.000, C 0.000 }
gfCNCPoint3[25031] = {X 281.9849, Y 16.1989, Z -4.6667, A 0.000, B 0.000, C 0.000 }
gfCNCPoint3[25032] = {X 281.3474, Y 15.5492, Z -4.6667, A 0.000, B 0.000, C 0.000 }
gfCNCPoint3[25033] = {X 280.8665, Y 14.7764, Z -4.6667, A 0.000, B 0.000, C 0.000 }
gfCNCPoint3[25034] = {X 280.5652, Y 13.9176, Z -4.6667, A 0.000, B 0.000, C 0.000 }
gfCNCPoint3[25035] = {X 280.4578, Y 13.0137, Z -4.6667, A 0.000, B 0.000, C 0.000 }
gfCNCPoint3[25036] = {X 280.4577, Y 12.1868, Z -4.6667, A 0.000, B 0.000, C 0.000 }
gfCNCPoint3[25037] = {X 280.5620, Y 11.2611, Z -4.6667, A 0.000, B 0.000, C 0.000 }
gfCNCPoint3[25038] = {X 280.8696, Y 10.3819, Z -4.6667, A 0.000, B 0.000, C 0.000 }
gfCNCPoint3[25039] = {X 281.3652, Y 9.5931, Z -4.6667, A 0.000, B 0.000, C 0.000 }
gfCNCPoint3[25040] = {X 282.0240, Y 8.9344, Z -4.6667, A 0.000, B 0.000, C 0.000 }
gfCNCPoint3[25041] = {X 282.8127, Y 8.4388, Z -4.6667, A 0.000, B 0.000, C 0.000 }
gfCNCPoint3[25042] = {X 283.6920, Y 8.1311, Z -4.6667, A 0.000, B 0.000, C 0.000 }
gfCNCPoint3[25043] = {X 284.6177, Y 8.0268, Z -4.6667, A 0.000, B 0.000, C 0.000 }
gfCNCPoint3[25044] = {X 291.0611, Y 8.0268, Z -4.6667, A 0.000, B 0.000, C 0.000 }
gfCNCPoint3[25045] = {X 291.9868, Y 8.1311, Z -4.6667, A 0.000, B 0.000, C 0.000 }
gfCNCPoint3[25046] = {X 292.8661, Y 8.4388, Z -4.6667, A 0.000, B 0.000, C 0.000 }
gfCNCPoint3[25047] = {X 293.6549, Y 8.9344, Z -4.6667, A 0.000, B 0.000, C 0.000 }
gfCNCPoint3[25048] = {X 294.3136, Y 9.5931, Z -4.6667, A 0.000, B 0.000, C 0.000 }
gfCNCPoint3[25049] = {X 294.8092, Y 10.3819, Z -4.6667, A 0.000, B 0.000, C 0.000 }
gfCNCPoint3[25050] = {X 295.1168, Y 11.2611, Z -4.6667, A 0.000, B 0.000, C 0.000 }
gfCNCPoint3[25051] = {X 295.2211, Y 12.1868, Z -4.6667, A 0.000, B 0.000, C 0.000 }
gfCNCPoint3[25052] = {X 295.2211, Y 12.9781, Z -4.6667, A 0.000, B 0.000, C 0.000 }
gfCNCPoint3[25053] = {X 295.1255, Y 13.8651, Z -4.6667, A 0.000, B 0.000, C 0.000 }
gfCNCPoint3[25054] = {X 294.8429, Y 14.7113, Z -4.6667, A 0.000, B 0.000, C 0.000 }
gfCNCPoint3[25055] = {X 294.3863, Y 15.4777, Z -4.6667, A 0.000, B 0.000, C 0.000 }
gfCNCPoint3[25056] = {X 293.7769, Y 16.1292, Z -4.6667, A 0.000, B 0.000, C 0.000 }
gfCNCPoint3[25057] = {X 293.6936, Y 16.1992, Z -4.6667, A 0.000, B 0.000, C 0.000 }
gfCNCPoint3[25058] = {X 293.6947, Y 22.3565, Z -4.6667, A 0.000, B 0.000, C 0.000 }
gfCNCPoint3[25059] = {X 302.9190, Y 22.3565, Z -4.6667, A 0.000, B 0.000, C 0.000 }
gfCNCPoint3[25060] = {X 302.9241, Y 16.2027, Z -4.6667, A 0.000, B 0.000, C 0.000 }
gfCNCPoint3[25061] = {X 302.2850, Y 15.5530, Z -4.6667, A 0.000, B 0.000, C 0.000 }
gfCNCPoint3[25062] = {X 301.8027, Y 14.7798, Z -4.6667, A 0.000, B 0.000, C 0.000 }
gfCNCPoint3[25063] = {X 301.5003, Y 13.9200, Z -4.6667, A 0.000, B 0.000, C 0.000 }
gfCNCPoint3[25064] = {X 301.3924, Y 13.0151, Z -4.6667, A 0.000, B 0.000, C 0.000 }
gfCNCPoint3[25065] = {X 301.3923, Y 12.1868, Z -4.6667, A 0.000, B 0.000, C 0.000 }
gfCNCPoint3[25066] = {X 301.4966, Y 11.2611, Z -4.6667, A 0.000, B 0.000, C 0.000 }
gfCNCPoint3[25067] = {X 301.8042, Y 10.3819, Z -4.6667, A 0.000, B 0.000, C 0.000 }
gfCNCPoint3[25068] = {X 302.2998, Y 9.5931, Z -4.6667, A 0.000, B 0.000, C 0.000 }
gfCNCPoint3[25069] = {X 302.9585, Y 8.9344, Z -4.6667, A 0.000, B 0.000, C 0.000 }
gfCNCPoint3[25070] = {X 303.7473, Y 8.4388, Z -4.6667, A 0.000, B 0.000, C 0.000 }
gfCNCPoint3[25071] = {X 304.6266, Y 8.1311, Z -4.6667, A 0.000, B 0.000, C 0.000 }
gfCNCPoint3[25072] = {X 305.5523, Y 8.0268, Z -4.6667, A 0.000, B 0.000, C 0.000 }
gfCNCPoint3[25073] = {X 311.9957, Y 8.0268, Z -4.6667, A 0.000, B 0.000, C 0.000 }
gfCNCPoint3[25074] = {X 312.9214, Y 8.1311, Z -4.6667, A 0.000, B 0.000, C 0.000 }
gfCNCPoint3[25075] = {X 313.8007, Y 8.4388, Z -4.6667, A 0.000, B 0.000, C 0.000 }
gfCNCPoint3[25076] = {X 314.5894, Y 8.9344, Z -4.6667, A 0.000, B 0.000, C 0.000 }
gfCNCPoint3[25077] = {X 315.2481, Y 9.5931, Z -4.6667, A 0.000, B 0.000, C 0.000 }
gfCNCPoint3[25078] = {X 315.7438, Y 10.3819, Z -4.6667, A 0.000, B 0.000, C 0.000 }
gfCNCPoint3[25079] = {X 316.0514, Y 11.2611, Z -4.6667, A 0.000, B 0.000, C 0.000 }
gfCNCPoint3[25080] = {X 316.1557, Y 12.1868, Z -4.6667, A 0.000, B 0.000, C 0.000 }
gfCNCPoint3[25081] = {X 316.1557, Y 12.9782, Z -4.6667, A 0.000, B 0.000, C 0.000 }
gfCNCPoint3[25082] = {X 316.0542, Y 13.8912, Z -4.6667, A 0.000, B 0.000, C 0.000 }
gfCNCPoint3[25083] = {X 315.7548, Y 14.7598, Z -4.6667, A 0.000, B 0.000, C 0.000 }
gfCNCPoint3[25084] = {X 315.2721, Y 15.5414, Z -4.6667, A 0.000, B 0.000, C 0.000 }
gfCNCPoint3[25085] = {X 314.6295, Y 16.1981, Z -4.6667, A 0.000, B 0.000, C 0.000 }
gfCNCPoint3[25086] = {X 314.6281, Y 40.9894, Z -4.6667, A 0.000, B 0.000, C 0.000 }
gfCNCPoint3[25087] = {X 314.6835, Y 41.0337, Z -4.6667, A 0.000, B 0.000, C 0.000 }
gfCNCPoint3[25088] = {X 315.2988, Y 41.6799, Z -4.6667, A 0.000, B 0.000, C 0.000 }
gfCNCPoint3[25089] = {X 315.7621, Y 42.4425, Z -4.6667, A 0.000, B 0.000, C 0.000 }
gfCNCPoint3[25090] = {X 316.0522, Y 43.2864, Z -4.6667, A 0.000, B 0.000, C 0.000 }
gfCNCPoint3[25091] = {X 316.1556, Y 44.1727, Z -4.6667, A 0.000, B 0.000, C 0.000 }
gfCNCPoint3[25092] = {X 316.1557, Y 45.0000, Z -4.6667, A 0.000, B 0.000, C 0.000 }
gfCNCPoint3[25093] = {X 316.0514, Y 45.9257, Z -4.6667, A 0.000, B 0.000, C 0.000 }
gfCNCPoint3[25094] = {X 315.7438, Y 46.8050, Z -4.6667, A 0.000, B 0.000, C 0.000 }
gfCNCPoint3[25095] = {X 315.2481, Y 47.5937, Z -4.6667, A 0.000, B 0.000, C 0.000 }
gfCNCPoint3[25096] = {X 314.5894, Y 48.2524, Z -4.6667, A 0.000, B 0.000, C 0.000 }
gfCNCPoint3[25097] = {X 313.8007, Y 48.7480, Z -4.6667, A 0.000, B 0.000, C 0.000 }
gfCNCPoint3[25098] = {X 312.9214, Y 49.0557, Z -4.6667, A 0.000, B 0.000, C 0.000 }
gfCNCPoint3[25099] = {X 311.9957, Y 49.1600, Z -4.6667, A 0.000, B 0.000, C 0.000 }
gfCNCPoint3[25100] = {X 305.5523, Y 49.1600, Z -4.6667, A 0.000, B 0.000, C 0.000 }
gfCNCPoint3[25101] = {X 304.6312, Y 49.0568, Z -4.6667, A 0.000, B 0.000, C 0.000 }
gfCNCPoint3[25102] = {X 303.7559, Y 48.7522, Z -4.6667, A 0.000, B 0.000, C 0.000 }
gfCNCPoint3[25103] = {X 302.9698, Y 48.2613, Z -4.6667, A 0.000, B 0.000, C 0.000 }
gfCNCPoint3[25104] = {X 302.3118, Y 47.6087, Z -4.6667, A 0.000, B 0.000, C 0.000 }
gfCNCPoint3[25105] = {X 301.8147, Y 46.8265, Z -4.6667, A 0.000, B 0.000, C 0.000 }
gfCNCPoint3[25106] = {X 301.5030, Y 45.9537, Z -4.6667, A 0.000, B 0.000, C 0.000 }
gfCNCPoint3[25107] = {X 301.3924, Y 45.0335, Z -4.6667, A 0.000, B 0.000, C 0.000 }
gfCNCPoint3[25108] = {X 301.3923, Y 44.2051, Z -4.6667, A 0.000, B 0.000, C 0.000 }
gfCNCPoint3[25109] = {X 301.5098, Y 43.2839, Z -4.6667, A 0.000, B 0.000, C 0.000 }
gfCNCPoint3[25110] = {X 301.8134, Y 42.4063, Z -4.6667, A 0.000, B 0.000, C 0.000 }
gfCNCPoint3[25111] = {X 302.2901, Y 41.6094, Z -4.6667, A 0.000, B 0.000, C 0.000 }
gfCNCPoint3[25112] = {X 302.9197, Y 40.9268, Z -4.6667, A 0.000, B 0.000, C 0.000 }
gfCNCPoint3[25113] = {X 302.9197, Y 33.8743, Z -4.6667, A 0.000, B 0.000, C 0.000 }
gfCNCPoint3[25114] = {X 293.6945, Y 33.8743, Z -4.6667, A 0.000, B 0.000, C 0.000 }
gfCNCPoint3[25115] = {X 293.6937, Y 40.9763, Z -4.6667, A 0.000, B 0.000, C 0.000 }
gfCNCPoint3[25116] = {X 294.3319, Y 41.6393, Z -4.6667, A 0.000, B 0.000, C 0.000 }
gfCNCPoint3[25117] = {X 294.8128, Y 42.4239, Z -4.6667, A 0.000, B 0.000, C 0.000 }
gfCNCPoint3[25118] = {X 295.1139, Y 43.2935, Z -4.6667, A 0.000, B 0.000, C 0.000 }
gfCNCPoint3[25119] = {X 295.2211, Y 44.2075, Z -4.6667, A 0.000, B 0.000, C 0.000 }
gfCNCPoint3[25120] = {X 295.2211, Y 45.0000, Z -4.6667, A 0.000, B 0.000, C 0.000 }
gfCNCPoint3[25121] = {X 295.1168, Y 45.9257, Z -4.6667, A 0.000, B 0.000, C 0.000 }
gfCNCPoint3[25122] = {X 294.8092, Y 46.8050, Z -4.6667, A 0.000, B 0.000, C 0.000 }
gfCNCPoint3[25123] = {X 294.3136, Y 47.5937, Z -4.6667, A 0.000, B 0.000, C 0.000 }
gfCNCPoint3[25124] = {X 293.6549, Y 48.2524, Z -4.6667, A 0.000, B 0.000, C 0.000 }
gfCNCPoint3[25125] = {X 292.8661, Y 48.7480, Z -4.6667, A 0.000, B 0.000, C 0.000 }
gfCNCPoint3[25126] = {X 291.9868, Y 49.0557, Z -4.6667, A 0.000, B 0.000, C 0.000 }
gfCNCPoint3[25127] = {X 291.0611, Y 49.1600, Z -4.6667, A 0.000, B 0.000, C 0.000 }
gfCNCPoint3[25128] = {X 284.6177, Y 49.1600, Z -4.6667, A 0.000, B 0.000, C 0.000 }
gfCNCPoint3[25129] = {X 283.6967, Y 49.0568, Z -4.6667, A 0.000, B 0.000, C 0.000 }
gfCNCPoint3[25130] = {X 282.8214, Y 48.7522, Z -4.6667, A 0.000, B 0.000, C 0.000 }
gfCNCPoint3[25131] = {X 282.0353, Y 48.2615, Z -4.6667, A 0.000, B 0.000, C 0.000 }
gfCNCPoint3[25132] = {X 281.3774, Y 47.6088, Z -4.6667, A 0.000, B 0.000, C 0.000 }
gfCNCPoint3[25133] = {X 280.8802, Y 46.8267, Z -4.6667, A 0.000, B 0.000, C 0.000 }
gfCNCPoint3[25134] = {X 280.5685, Y 45.9540, Z -4.6667, A 0.000, B 0.000, C 0.000 }
gfCNCPoint3[25135] = {X 280.4578, Y 45.0339, Z -4.6667, A 0.000, B 0.000, C 0.000 }
gfCNCPoint3[25136] = {X 280.4577, Y 44.2081, Z -4.6667, A 0.000, B 0.000, C 0.000 }
gfCNCPoint3[25137] = {X 280.5627, Y 43.2952, Z -4.6667, A 0.000, B 0.000, C 0.000 }
gfCNCPoint3[25138] = {X 280.8633, Y 42.4269, Z -4.6667, A 0.000, B 0.000, C 0.000 }
gfCNCPoint3[25139] = {X 281.3451, Y 41.6445, Z -4.6667, A 0.000, B 0.000, C 0.000 }
gfCNCPoint3[25140] = {X 281.9853, Y 40.9854, Z -4.6667, A 0.000, B 0.000, C 0.000 }
gfCNCPoint3[25141] = {X 281.9851, Y 28.5924, Z -4.6667, A 0.000, B 0.000, C 0.000 }
gfCNCPoint3[25142] = {X 277.9851, Y 28.5925, Z -4.6667, A 0.000, B 0.000, C 0.000 }
gfCNCPoint3[25143] = {X 282.0651, Y 28.5924, Z -4.6667, A 0.000, B 0.000, C 0.000 }
gfCNCPoint3[25144] = {X 282.0649, Y 16.1608, Z -4.6667, A 0.000, B 0.000, C 0.000 }
gfCNCPoint3[25145] = {X 281.4279, Y 15.5220, Z -4.6667, A 0.000, B 0.000, C 0.000 }
gfCNCPoint3[25146] = {X 280.9468, Y 14.7589, Z -4.6667, A 0.000, B 0.000, C 0.000 }
gfCNCPoint3[25147] = {X 280.6452, Y 13.9087, Z -4.6667, A 0.000, B 0.000, C 0.000 }
gfCNCPoint3[25148] = {X 280.5378, Y 13.0130, Z -4.6667, A 0.000, B 0.000, C 0.000 }
gfCNCPoint3[25149] = {X 280.5377, Y 12.1868, Z -4.6667, A 0.000, B 0.000, C 0.000 }
gfCNCPoint3[25150] = {X 280.6400, Y 11.2789, Z -4.6667, A 0.000, B 0.000, C 0.000 }
gfCNCPoint3[25151] = {X 280.9417, Y 10.4166, Z -4.6667, A 0.000, B 0.000, C 0.000 }
gfCNCPoint3[25152] = {X 281.4278, Y 9.6430, Z -4.6667, A 0.000, B 0.000, C 0.000 }
gfCNCPoint3[25153] = {X 282.0738, Y 8.9969, Z -4.6667, A 0.000, B 0.000, C 0.000 }
gfCNCPoint3[25154] = {X 282.8474, Y 8.5109, Z -4.6667, A 0.000, B 0.000, C 0.000 }
gfCNCPoint3[25155] = {X 283.7098, Y 8.2091, Z -4.6667, A 0.000, B 0.000, C 0.000 }
gfCNCPoint3[25156] = {X 284.6177, Y 8.1068, Z -4.6667, A 0.000, B 0.000, C 0.000 }
gfCNCPoint3[25157] = {X 291.0611, Y 8.1068, Z -4.6667, A 0.000, B 0.000, C 0.000 }
gfCNCPoint3[25158] = {X 291.9690, Y 8.2091, Z -4.6667, A 0.000, B 0.000, C 0.000 }
gfCNCPoint3[25159] = {X 292.8314, Y 8.5109, Z -4.6667, A 0.000, B 0.000, C 0.000 }
gfCNCPoint3[25160] = {X 293.6050, Y 8.9969, Z -4.6667, A 0.000, B 0.000, C 0.000 }
gfCNCPoint3[25161] = {X 294.2510, Y 9.6430, Z -4.6667, A 0.000, B 0.000, C 0.000 }
gfCNCPoint3[25162] = {X 294.7371, Y 10.4166, Z -4.6667, A 0.000, B 0.000, C 0.000 }
gfCNCPoint3[25163] = {X 295.0388, Y 11.2789, Z -4.6667, A 0.000, B 0.000, C 0.000 }
gfCNCPoint3[25164] = {X 295.1411, Y 12.1868, Z -4.6667, A 0.000, B 0.000, C 0.000 }
gfCNCPoint3[25165] = {X 295.1411, Y 12.9781, Z -4.6667, A 0.000, B 0.000, C 0.000 }
gfCNCPoint3[25166] = {X 295.0473, Y 13.8481, Z -4.6667, A 0.000, B 0.000, C 0.000 }
gfCNCPoint3[25167] = {X 294.7701, Y 14.6780, Z -4.6667, A 0.000, B 0.000, C 0.000 }
gfCNCPoint3[25168] = {X 294.3224, Y 15.4297, Z -4.6667, A 0.000, B 0.000, C 0.000 }
gfCNCPoint3[25169] = {X 293.7247, Y 16.0686, Z -4.6667, A 0.000, B 0.000, C 0.000 }
gfCNCPoint3[25170] = {X 293.6672, Y 16.1172, Z -4.6667, A 0.000, B 0.000, C 0.000 }
gfCNCPoint3[25171] = {X 293.6089, Y 16.1647, Z -4.6667, A 0.000, B 0.000, C 0.000 }
gfCNCPoint3[25172] = {X 293.6136, Y 16.1992, Z -4.6667, A 0.000, B 0.000, C 0.000 }
gfCNCPoint3[25173] = {X 293.6147, Y 22.4366, Z -4.6667, A 0.000, B 0.000, C 0.000 }
gfCNCPoint3[25174] = {X 293.7676, Y 22.4365, Z -4.6667, A 0.000, B 0.000, C 0.000 }
gfCNCPoint3[25175] = {X 302.9989, Y 22.4365, Z -4.6667, A 0.000, B 0.000, C 0.000 }
gfCNCPoint3[25176] = {X 303.0042, Y 16.1645, Z -4.6667, A 0.000, B 0.000, C 0.000 }
gfCNCPoint3[25177] = {X 302.9458, Y 16.1169, Z -4.6667, A 0.000, B 0.000, C 0.000 }
gfCNCPoint3[25178] = {X 302.8883, Y 16.0683, Z -4.6667, A 0.000, B 0.000, C 0.000 }
gfCNCPoint3[25179] = {X 302.2962, Y 15.4366, Z -4.6667, A 0.000, B 0.000, C 0.000 }
gfCNCPoint3[25180] = {X 301.8507, Y 14.6942, Z -4.6667, A 0.000, B 0.000, C 0.000 }
gfCNCPoint3[25181] = {X 301.5720, Y 13.8745, Z -4.6667, A 0.000, B 0.000, C 0.000 }
gfCNCPoint3[25182] = {X 301.4724, Y 13.0144, Z -4.6667, A 0.000, B 0.000, C 0.000 }
gfCNCPoint3[25183] = {X 301.4723, Y 12.1868, Z -4.6667, A 0.000, B 0.000, C 0.000 }
gfCNCPoint3[25184] = {X 301.5745, Y 11.2789, Z -4.6667, A 0.000, B 0.000, C 0.000 }
gfCNCPoint3[25185] = {X 301.8763, Y 10.4166, Z -4.6667, A 0.000, B 0.000, C 0.000 }
gfCNCPoint3[25186] = {X 302.3624, Y 9.6430, Z -4.6667, A 0.000, B 0.000, C 0.000 }
gfCNCPoint3[25187] = {X 303.0084, Y 8.9969, Z -4.6667, A 0.000, B 0.000, C 0.000 }
gfCNCPoint3[25188] = {X 303.7820, Y 8.5109, Z -4.6667, A 0.000, B 0.000, C 0.000 }
gfCNCPoint3[25189] = {X 304.6444, Y 8.2091, Z -4.6667, A 0.000, B 0.000, C 0.000 }
gfCNCPoint3[25190] = {X 305.5523, Y 8.1068, Z -4.6667, A 0.000, B 0.000, C 0.000 }
gfCNCPoint3[25191] = {X 311.9957, Y 8.1068, Z -4.6667, A 0.000, B 0.000, C 0.000 }
gfCNCPoint3[25192] = {X 312.9036, Y 8.2091, Z -4.6667, A 0.000, B 0.000, C 0.000 }
gfCNCPoint3[25193] = {X 313.7660, Y 8.5109, Z -4.6667, A 0.000, B 0.000, C 0.000 }
gfCNCPoint3[25194] = {X 314.5396, Y 8.9969, Z -4.6667, A 0.000, B 0.000, C 0.000 }
gfCNCPoint3[25195] = {X 315.1856, Y 9.6430, Z -4.6667, A 0.000, B 0.000, C 0.000 }
gfCNCPoint3[25196] = {X 315.6717, Y 10.4166, Z -4.6667, A 0.000, B 0.000, C 0.000 }
gfCNCPoint3[25197] = {X 315.9734, Y 11.2789, Z -4.6667, A 0.000, B 0.000, C 0.000 }
gfCNCPoint3[25198] = {X 316.0757, Y 12.1868, Z -4.6667, A 0.000, B 0.000, C 0.000 }
gfCNCPoint3[25199] = {X 316.0757, Y 12.9782, Z -4.6667, A 0.000, B 0.000, C 0.000 }
gfCNCPoint3[25200] = {X 315.9741, Y 13.8829, Z -4.6667, A 0.000, B 0.000, C 0.000 }
